LIN {X -0.054,Y -673.462,Z 1135.531,A 0.000,B 0.000,C 90.000,E1 131.595} C_DIS
LIN {X -0.295,Y -677.512,Z 1135.522,A 0.000,B 0.000,C 90.000,E1 129.930} C_DIS
LIN {X -0.323,Y -682.386,Z 1135.511,A 0.000,B 0.000,C 90.000,E1 128.016} C_DIS
LIN {X 0.074,Y -685.376,Z 1135.505,A 0.000,B 0.000,C 90.000,E1 126.790} C_DIS
LIN {X -0.070,Y -687.830,Z 1135.499,A 0.000,B 0.000,C 90.000,E1 125.851} C_DIS
LIN {X 0.211,Y -691.281,Z 1135.491,A 0.000,B 0.000,C 90.000,E1 124.405} C_DIS
LIN {X -0.010,Y -694.725,Z 1135.483,A 0.000,B 0.000,C 90.000,E1 123.007} C_DIS
LIN {X 0.378,Y -697.379,Z 1135.477,A 0.000,B 0.000,C 90.000,E1 121.799} C_DIS
LIN {X 0.197,Y -699.151,Z 1135.472,A 0.000,B 0.000,C 90.000,E1 120.875} C_DIS
LIN {X -0.296,Y -701.217,Z 1135.465,A 0.000,B 0.000,C 90.000,E1 119.745} C_DIS
LIN {X 0.133,Y -703.611,Z 1135.457,A 0.000,B 0.000,C 90.000,E1 118.309} C_DIS
LIN {X -0.259,Y -704.683,Z 1135.453,A 0.000,B 0.000,C 90.000,E1 117.641} C_DIS
LIN {X -0.025,Y -705.467,Z 1135.450,A 0.000,B 0.000,C 90.000,E1 116.924} C_DIS
LIN {X -0.153,Y -706.164,Z 1135.443,A 0.000,B 0.000,C 90.000,E1 115.771} C_DIS
LIN {X -0.220,Y -706.290,Z 1135.439,A 0.000,B 0.000,C 90.000,E1 115.079} C_DIS
LIN {X 0.068,Y -706.168,Z 1135.437,A 0.000,B 0.000,C 90.000,E1 114.591} C_DIS
LIN {X 0.006,Y -705.430,Z 1135.434,A 0.000,B 0.000,C 90.000,E1 114.131} C_DIS
LIN {X 0.008,Y -704.956,Z 1135.433,A 0.000,B 0.000,C 90.000,E1 113.898} C_DIS
LIN {X -0.206,Y -702.429,Z 1135.430,A 0.000,B 0.000,C 90.000,E1 113.334} C_DIS
LIN {X -0.066,Y -701.628,Z 1135.429,A 0.000,B 0.000,C 90.000,E1 113.206} C_DIS
LIN {X 0.201,Y -697.281,Z 1135.426,A 0.000,B 0.000,C 90.000,E1 112.717} C_DIS
LIN {X -0.312,Y -695.828,Z 1135.426,A 0.000,B 0.000,C 90.000,E1 112.642} C_DIS
LIN {X -0.182,Y -693.351,Z 1135.425,A 0.000,B 0.000,C 90.000,E1 112.514} C_DIS
LIN {X 0.282,Y -685.424,Z 1135.424,A 0.000,B 0.000,C 90.000,E1 112.206} C_DIS
LIN {X -0.173,Y -682.533,Z 1135.423,A 0.000,B 0.000,C 90.000,E1 112.206} C_DIS
LIN {X -0.220,Y -676.235,Z 1135.423,A 0.000,B 0.000,C 90.000,E1 112.153} C_DIS
LIN {X -0.243,Y -603.153,Z 1135.423,A 0.000,B 0.000,C 90.000,E1 112.153} C_DIS
LIN {X 0.311,Y -600.036,Z 1135.422,A 0.000,B 0.000,C 90.000,E1 111.897} C_DIS
LIN {X -0.184,Y -595.483,Z 1135.420,A 0.000,B 0.000,C 90.000,E1 111.589} C_DIS
LIN {X -0.037,Y -584.010,Z 1135.414,A 0.000,B 0.000,C 90.000,E1 110.556} C_DIS
LIN {X 0.171,Y -575.780,Z 1135.410,A 0.000,B 0.000,C 90.000,E1 109.812} C_DIS
LIN {X -0.325,Y -569.798,Z 1135.408,A 0.000,B 0.000,C 90.000,E1 109.396} C_DIS
LIN {X -0.170,Y -568.295,Z 1135.407,A 0.000,B 0.000,C 90.000,E1 109.268} C_DIS
LIN {X 0.057,Y -560.118,Z 1135.404,A 0.000,B 0.000,C 90.000,E1 108.725} C_DIS
LIN {X 0.230,Y -555.289,Z 1135.402,A 0.000,B 0.000,C 90.000,E1 108.417} C_DIS
LIN {X -0.209,Y -550.970,Z 1135.401,A 0.000,B 0.000,C 90.000,E1 108.127} C_DIS
LIN {X 0.260,Y -549.678,Z 1135.400,A 0.000,B 0.000,C 90.000,E1 107.873} C_DIS
LIN {X 0.219,Y -549.656,Z 1135.399,A 0.000,B 0.000,C 90.000,E1 107.873} C_DIS
LIN {X 0.011,Y -549.420,Z 1135.397,A 0.000,B 0.000,C 90.000,E1 107.457} C_DIS
LIN {X 0.002,Y -551.243,Z 1135.381,A 0.000,B 0.000,C 90.000,E1 104.662} C_DIS
LIN {X -0.248,Y -552.639,Z 1135.372,A 0.000,B 0.000,C 90.000,E1 103.008} C_DIS
LIN {X 0.058,Y -554.057,Z 1135.363,A 0.000,B 0.000,C 90.000,E1 101.299} C_DIS
LIN {X 0.043,Y -555.316,Z 1135.355,A 0.000,B 0.000,C 90.000,E1 99.905} C_DIS
LIN {X 0.186,Y -556.857,Z 1135.346,A 0.000,B 0.000,C 90.000,E1 98.219} C_DIS
LIN {X 0.142,Y -558.055,Z 1135.338,A 0.000,B 0.000,C 90.000,E1 96.834} C_DIS
LIN {X 0.193,Y -559.539,Z 1135.329,A 0.000,B 0.000,C 90.000,E1 95.163} C_DIS
LIN {X 0.140,Y -560.678,Z 1135.321,A 0.000,B 0.000,C 90.000,E1 93.784} C_DIS
LIN {X 0.072,Y -561.691,Z 1135.313,A 0.000,B 0.000,C 90.000,E1 92.407} C_DIS
LIN {X 0.022,Y -562.668,Z 1135.306,A 0.000,B 0.000,C 90.000,E1 91.031} C_DIS
LIN {X 0.081,Y -563.758,Z 1135.297,A 0.000,B 0.000,C 90.000,E1 89.370} C_DIS
LIN {X -0.164,Y -564.194,Z 1135.292,A 0.000,B 0.000,C 90.000,E1 88.568} C_DIS
LIN {X -0.067,Y -565.185,Z 1135.283,A 0.000,B 0.000,C 90.000,E1 86.906} C_DIS
LIN {X -0.026,Y -565.914,Z 1135.275,A 0.000,B 0.000,C 90.000,E1 85.527} C_DIS
LIN {X 0.031,Y -566.496,Z 1135.268,A 0.000,B 0.000,C 90.000,E1 84.147} C_DIS
LIN {X -0.236,Y -567.248,Z 1135.258,A 0.000,B 0.000,C 90.000,E1 82.527} C_DIS
LIN {X -0.092,Y -567.901,Z 1135.251,A 0.000,B 0.000,C 90.000,E1 81.141} C_DIS
LIN {X -0.235,Y -568.620,Z 1135.242,A 0.000,B 0.000,C 90.000,E1 79.511} C_DIS
LIN {X -0.186,Y -569.504,Z 1135.231,A 0.000,B 0.000,C 90.000,E1 77.589} C_DIS
LIN {X -0.063,Y -570.280,Z 1135.222,A 0.000,B 0.000,C 90.000,E1 75.936} C_DIS
LIN {X 0.045,Y -571.479,Z 1135.210,A 0.000,B 0.000,C 90.000,E1 73.740} C_DIS
LIN {X 0.181,Y -572.362,Z 1135.202,A 0.000,B 0.000,C 90.000,E1 72.362} C_DIS
LIN {X 0.142,Y -573.611,Z 1135.193,A 0.000,B 0.000,C 90.000,E1 70.732} C_DIS
LIN {X 0.152,Y -575.711,Z 1135.179,A 0.000,B 0.000,C 90.000,E1 68.284} C_DIS
LIN {X 0.208,Y -577.022,Z 1135.172,A 0.000,B 0.000,C 90.000,E1 66.922} C_DIS
LIN {X 0.130,Y -578.428,Z 1135.163,A 0.000,B 0.000,C 90.000,E1 65.305} C_DIS
LIN {X -0.306,Y -579.211,Z 1135.158,A 0.000,B 0.000,C 90.000,E1 64.537} C_DIS
LIN {X 0.151,Y -580.566,Z 1135.149,A 0.000,B 0.000,C 90.000,E1 62.871} C_DIS
LIN {X 0.119,Y -581.934,Z 1135.140,A 0.000,B 0.000,C 90.000,E1 61.257} C_DIS
LIN {X -0.114,Y -583.067,Z 1135.131,A 0.000,B 0.000,C 90.000,E1 59.665} C_DIS
LIN {X -0.189,Y -583.979,Z 1135.124,A 0.000,B 0.000,C 90.000,E1 58.329} C_DIS
LIN {X -0.078,Y -584.923,Z 1135.115,A 0.000,B 0.000,C 90.000,E1 56.707} C_DIS
LIN {X -0.113,Y -585.846,Z 1135.106,A 0.000,B 0.000,C 90.000,E1 55.102} C_DIS
LIN {X -0.131,Y -586.745,Z 1135.097,A 0.000,B 0.000,C 90.000,E1 53.497} C_DIS
LIN {X -0.019,Y -587.109,Z 1135.093,A 0.000,B 0.000,C 90.000,E1 52.683} C_DIS
LIN {X 0.064,Y -587.974,Z 1135.082,A 0.000,B 0.000,C 90.000,E1 50.803} C_DIS
LIN {X -0.061,Y -588.254,Z 1135.076,A 0.000,B 0.000,C 90.000,E1 49.747} C_DIS
LIN {X -0.179,Y -588.386,Z 1135.070,A 0.000,B 0.000,C 90.000,E1 48.690} C_DIS
LIN {X 0.216,Y -588.248,Z 1135.060,A 0.000,B 0.000,C 90.000,E1 46.782} C_DIS
LIN {X -0.188,Y -587.888,Z 1135.053,A 0.000,B 0.000,C 90.000,E1 45.486} C_DIS
LIN {X -0.345,Y -587.498,Z 1135.047,A 0.000,B 0.000,C 90.000,E1 44.433} C_DIS
LIN {X -0.086,Y -586.841,Z 1135.041,A 0.000,B 0.000,C 90.000,E1 43.338} C_DIS
LIN {X 0.242,Y -586.545,Z 1135.038,A 0.000,B 0.000,C 90.000,E1 42.771} C_DIS
LIN {X 0.169,Y -585.976,Z 1135.035,A 0.000,B 0.000,C 90.000,E1 42.243} C_DIS
LIN {X -0.086,Y -585.834,Z 1135.033,A 0.000,B 0.000,C 90.000,E1 42.000} C_DIS
LIN {X 0.058,Y -583.950,Z 1135.024,A 0.000,B 0.000,C 90.000,E1 40.378} C_DIS
LIN {X -0.033,Y -583.350,Z 1135.021,A 0.000,B 0.000,C 90.000,E1 39.850} C_DIS
LIN {X -0.059,Y -581.407,Z 1135.014,A 0.000,B 0.000,C 90.000,E1 38.508} C_DIS
LIN {X -0.023,Y -579.036,Z 1135.006,A 0.000,B 0.000,C 90.000,E1 37.156} C_DIS
LIN {X -0.339,Y -577.328,Z 1135.002,A 0.000,B 0.000,C 90.000,E1 36.377} C_DIS
LIN {X 0.134,Y -575.314,Z 1134.997,A 0.000,B 0.000,C 90.000,E1 35.518} C_DIS
LIN {X 0.103,Y -573.841,Z 1134.994,A 0.000,B 0.000,C 90.000,E1 34.978} C_DIS
LIN {X -0.265,Y -571.310,Z 1134.990,A 0.000,B 0.000,C 90.000,E1 34.199} C_DIS
LIN {X 0.001,Y -569.465,Z 1134.987,A 0.000,B 0.000,C 90.000,E1 33.627} C_DIS
LIN {X -0.142,Y -565.241,Z 1134.981,A 0.000,B 0.000,C 90.000,E1 32.546} C_DIS
LIN {X -0.331,Y -562.292,Z 1134.977,A 0.000,B 0.000,C 90.000,E1 31.878} C_DIS
LIN {X 0.190,Y -556.954,Z 1134.971,A 0.000,B 0.000,C 90.000,E1 30.718} C_DIS
LIN {X 0.176,Y -551.709,Z 1134.965,A 0.000,B 0.000,C 90.000,E1 29.745} C_DIS
LIN {X -0.254,Y -546.846,Z 1134.961,A 0.000,B 0.000,C 90.000,E1 28.949} C_DIS
LIN {X 0.094,Y -540.592,Z 1134.955,A 0.000,B 0.000,C 90.000,E1 27.924} C_DIS
LIN {X 0.024,Y -534.510,Z 1134.950,A 0.000,B 0.000,C 90.000,E1 27.078} C_DIS
LIN {X 0.033,Y -529.067,Z 1134.947,A 0.000,B 0.000,C 90.000,E1 26.360} C_DIS
LIN {X -0.208,Y -523.297,Z 1134.943,A 0.000,B 0.000,C 90.000,E1 25.668} C_DIS
LIN {X -0.110,Y -514.407,Z 1134.937,A 0.000,B 0.000,C 90.000,E1 24.643} C_DIS
LIN {X 0.110,Y -507.754,Z 1134.933,A 0.000,B 0.000,C 90.000,E1 23.898} C_DIS
LIN {X -0.063,Y -499.557,Z 1134.928,A 0.000,B 0.000,C 90.000,E1 23.078} C_DIS
LIN {X -0.207,Y -491.090,Z 1134.924,A 0.000,B 0.000,C 90.000,E1 22.280} C_DIS
LIN {X 0.040,Y -483.962,Z 1134.920,A 0.000,B 0.000,C 90.000,E1 21.589} C_DIS
LIN {X 0.239,Y -475.392,Z 1134.916,A 0.000,B 0.000,C 90.000,E1 20.791} C_DIS
LIN {X -0.073,Y -468.011,Z 1134.912,A 0.000,B 0.000,C 90.000,E1 20.174} C_DIS
LIN {X 0.109,Y -453.457,Z 1134.905,A 0.000,B 0.000,C 90.000,E1 18.852} C_DIS
LIN {X 0.049,Y -437.348,Z 1134.896,A 0.000,B 0.000,C 90.000,E1 17.347} C_DIS
LIN {X -0.102,Y -423.156,Z 1134.888,A 0.000,B 0.000,C 90.000,E1 15.898} C_DIS
LIN {X 0.159,Y -412.057,Z 1134.881,A 0.000,B 0.000,C 90.000,E1 14.592} C_DIS
LIN {X 0.188,Y -404.239,Z 1134.876,A 0.000,B 0.000,C 90.000,E1 13.592} C_DIS
LIN {X 0.056,Y -399.562,Z 1134.872,A 0.000,B 0.000,C 90.000,E1 12.939} C_DIS
LIN {X 0.041,Y -397.373,Z 1134.870,A 0.000,B 0.000,C 90.000,E1 12.591} C_DIS
LIN {X -0.181,Y -394.183,Z 1134.867,A 0.000,B 0.000,C 90.000,E1 12.007} C_DIS
LIN {X 0.121,Y -392.964,Z 1134.865,A 0.000,B 0.000,C 90.000,E1 11.591} C_DIS
LIN {X 0.063,Y -392.555,Z 1134.864,A 0.000,B 0.000,C 90.000,E1 11.422} C_DIS
LIN {X 0.051,Y -392.145,Z 1134.862,A 0.000,B 0.000,C 90.000,E1 11.074} C_DIS
LIN {X 0.065,Y -392.473,Z 1134.859,A 0.000,B 0.000,C 90.000,E1 10.546} C_DIS
LIN {X 0.077,Y -392.640,Z 1134.858,A 0.000,B 0.000,C 90.000,E1 10.366} C_DIS
LIN {X -0.078,Y -394.573,Z 1134.852,A 0.000,B 0.000,C 90.000,E1 9.434} C_DIS
LIN {X 0.146,Y -397.451,Z 1134.847,A 0.000,B 0.000,C 90.000,E1 8.341} C_DIS
LIN {X -0.003,Y -402.854,Z 1134.837,A 0.000,B 0.000,C 90.000,E1 6.606} C_DIS
LIN {X -0.036,Y -404.749,Z 1134.834,A 0.000,B 0.000,C 90.000,E1 6.087} C_DIS
LIN {X -0.057,Y -407.334,Z 1134.831,A 0.000,B 0.000,C 90.000,E1 5.568} C_DIS
LIN {X -0.034,Y -408.383,Z 1134.830,A 0.000,B 0.000,C 90.000,E1 5.391} C_DIS
LIN {X -0.051,Y -411.120,Z 1134.828,A 0.000,B 0.000,C 90.000,E1 5.049} C_DIS
LIN {X -0.052,Y -412.815,Z 1134.827,A 0.000,B 0.000,C 90.000,E1 4.878} C_DIS
LIN {X -0.122,Y -416.366,Z 1134.825,A 0.000,B 0.000,C 90.000,E1 4.588} C_DIS
LIN {X 0.180,Y -423.924,Z 1134.823,A 0.000,B 0.000,C 90.000,E1 4.012} C_DIS
LIN {X 0.208,Y -446.765,Z 1134.814,A 0.000,B 0.000,C 90.000,E1 2.407} C_DIS
LIN {X 0.220,Y -463.099,Z 1134.807,A 0.000,B 0.000,C 90.000,E1 1.318} C_DIS
LIN {X -0.195,Y -474.343,Z 1134.803,A 0.000,B 0.000,C 90.000,E1 0.630} C_DIS
LIN {X 0.000,Y -483.330,Z 1134.800,A 0.000,B 0.000,C 90.000,E1 360.000} C_DIS
LIN {X 0.238,Y -490.911,Z 1134.797,A 0.000,B 0.000,C 90.000,E1 359.427} C_DIS
LIN {X -0.246,Y -496.999,Z 1134.794,A 0.000,B 0.000,C 90.000,E1 359.026} C_DIS
LIN {X 0.117,Y -502.993,Z 1134.792,A 0.000,B 0.000,C 90.000,E1 358.511} C_DIS
LIN {X 0.177,Y -510.196,Z 1134.788,A 0.000,B 0.000,C 90.000,E1 357.879} C_DIS
LIN {X 0.038,Y -517.140,Z 1134.785,A 0.000,B 0.000,C 90.000,E1 357.249} C_DIS
LIN {X 0.060,Y -521.102,Z 1134.783,A 0.000,B 0.000,C 90.000,E1 356.846} C_DIS
LIN {X -0.041,Y -527.440,Z 1134.779,A 0.000,B 0.000,C 90.000,E1 356.159} C_DIS
LIN {X 0.024,Y -532.263,Z 1134.776,A 0.000,B 0.000,C 90.000,E1 355.584} C_DIS
LIN {X -0.240,Y -537.755,Z 1134.771,A 0.000,B 0.000,C 90.000,E1 354.894} C_DIS
LIN {X 0.081,Y -542.573,Z 1134.768,A 0.000,B 0.000,C 90.000,E1 354.147} C_DIS
LIN {X -0.035,Y -546.969,Z 1134.764,A 0.000,B 0.000,C 90.000,E1 353.451} C_DIS
LIN {X 0.084,Y -550.174,Z 1134.760,A 0.000,B 0.000,C 90.000,E1 352.875} C_DIS
LIN {X 0.088,Y -555.222,Z 1134.755,A 0.000,B 0.000,C 90.000,E1 351.894} C_DIS
LIN {X -0.292,Y -557.758,Z 1134.752,A 0.000,B 0.000,C 90.000,E1 351.376} C_DIS
LIN {X -0.269,Y -560.636,Z 1134.748,A 0.000,B 0.000,C 90.000,E1 350.679} C_DIS
LIN {X 0.181,Y -563.777,Z 1134.744,A 0.000,B 0.000,C 90.000,E1 349.803} C_DIS
LIN {X 0.011,Y -566.665,Z 1134.739,A 0.000,B 0.000,C 90.000,E1 348.993} C_DIS
LIN {X 0.156,Y -570.210,Z 1134.733,A 0.000,B 0.000,C 90.000,E1 347.881} C_DIS
LIN {X 0.119,Y -574.235,Z 1134.725,A 0.000,B 0.000,C 90.000,E1 346.520} C_DIS
LIN {X 0.018,Y -577.923,Z 1134.718,A 0.000,B 0.000,C 90.000,E1 345.172} C_DIS
LIN {X 0.275,Y -581.457,Z 1134.710,A 0.000,B 0.000,C 90.000,E1 343.795} C_DIS
LIN {X 0.271,Y -585.478,Z 1134.701,A 0.000,B 0.000,C 90.000,E1 342.181} C_DIS
LIN {X 0.016,Y -587.351,Z 1134.697,A 0.000,B 0.000,C 90.000,E1 341.402} C_DIS
LIN {X 0.197,Y -589.644,Z 1134.691,A 0.000,B 0.000,C 90.000,E1 340.315} C_DIS
LIN {X 0.058,Y -591.720,Z 1134.685,A 0.000,B 0.000,C 90.000,E1 339.263} C_DIS
LIN {X -0.263,Y -593.666,Z 1134.679,A 0.000,B 0.000,C 90.000,E1 338.230} C_DIS
LIN {X -0.016,Y -594.827,Z 1134.675,A 0.000,B 0.000,C 90.000,E1 337.411} C_DIS
LIN {X -0.167,Y -596.352,Z 1134.667,A 0.000,B 0.000,C 90.000,E1 336.102} C_DIS
LIN {X -0.216,Y -597.148,Z 1134.661,A 0.000,B 0.000,C 90.000,E1 335.049} C_DIS
LIN {X 0.072,Y -597.559,Z 1134.657,A 0.000,B 0.000,C 90.000,E1 334.229} C_DIS
LIN {X 0.093,Y -597.595,Z 1134.652,A 0.000,B 0.000,C 90.000,E1 333.435} C_DIS
LIN {X -0.145,Y -597.263,Z 1134.648,A 0.000,B 0.000,C 90.000,E1 332.666} C_DIS
LIN {X 0.137,Y -596.685,Z 1134.644,A 0.000,B 0.000,C 90.000,E1 331.847} C_DIS
LIN {X 0.252,Y -596.143,Z 1134.641,A 0.000,B 0.000,C 90.000,E1 331.307} C_DIS
LIN {X -0.012,Y -595.032,Z 1134.636,A 0.000,B 0.000,C 90.000,E1 330.539} C_DIS
LIN {X 0.203,Y -592.887,Z 1134.630,A 0.000,B 0.000,C 90.000,E1 329.459} C_DIS
LIN {X -0.001,Y -591.481,Z 1134.628,A 0.000,B 0.000,C 90.000,E1 328.948} C_DIS
LIN {X 0.087,Y -589.792,Z 1134.625,A 0.000,B 0.000,C 90.000,E1 328.408} C_DIS
LIN {X 0.164,Y -587.964,Z 1134.622,A 0.000,B 0.000,C 90.000,E1 327.867} C_DIS
LIN {X -0.076,Y -584.644,Z 1134.617,A 0.000,B 0.000,C 90.000,E1 327.089} C_DIS
LIN {X -0.107,Y -581.397,Z 1134.613,A 0.000,B 0.000,C 90.000,E1 326.421} C_DIS
LIN {X 0.070,Y -576.825,Z 1134.609,A 0.000,B 0.000,C 90.000,E1 325.595} C_DIS
LIN {X 0.048,Y -573.585,Z 1134.606,A 0.000,B 0.000,C 90.000,E1 325.055} C_DIS
LIN {X -0.232,Y -569.139,Z 1134.602,A 0.000,B 0.000,C 90.000,E1 324.402} C_DIS
LIN {X -0.205,Y -566.307,Z 1134.600,A 0.000,B 0.000,C 90.000,E1 323.989} C_DIS
LIN {X 0.027,Y -562.124,Z 1134.597,A 0.000,B 0.000,C 90.000,E1 323.417} C_DIS
LIN {X -0.254,Y -554.221,Z 1134.591,A 0.000,B 0.000,C 90.000,E1 322.477} C_DIS
LIN {X -0.053,Y -546.776,Z 1134.587,A 0.000,B 0.000,C 90.000,E1 321.618} C_DIS
LIN {X -0.142,Y -536.796,Z 1134.581,A 0.000,B 0.000,C 90.000,E1 320.517} C_DIS
LIN {X -0.018,Y -533.738,Z 1134.578,A 0.000,B 0.000,C 90.000,E1 320.114} C_DIS
LIN {X 0.064,Y -530.380,Z 1134.576,A 0.000,B 0.000,C 90.000,E1 319.585} C_DIS
LIN {X -0.124,Y -527.923,Z 1134.573,A 0.000,B 0.000,C 90.000,E1 319.094} C_DIS
LIN {X -0.183,Y -526.213,Z 1134.570,A 0.000,B 0.000,C 90.000,E1 318.609} C_DIS
LIN {X 0.088,Y -525.373,Z 1134.568,A 0.000,B 0.000,C 90.000,E1 318.243} C_DIS
LIN {X -0.190,Y -524.466,Z 1134.566,A 0.000,B 0.000,C 90.000,E1 317.838} C_DIS
LIN {X 0.222,Y -523.768,Z 1134.562,A 0.000,B 0.000,C 90.000,E1 317.067} C_DIS
LIN {X 0.338,Y -523.606,Z 1134.555,A 0.000,B 0.000,C 90.000,E1 315.891} C_DIS
LIN {X -0.056,Y -523.818,Z 1134.546,A 0.000,B 0.000,C 90.000,E1 314.190} C_DIS
LIN {X 0.182,Y -524.344,Z 1134.533,A 0.000,B 0.000,C 90.000,E1 311.838} C_DIS
LIN {X -0.264,Y -525.395,Z 1134.520,A 0.000,B 0.000,C 90.000,E1 309.564} C_DIS
LIN {X -0.198,Y -526.773,Z 1134.507,A 0.000,B 0.000,C 90.000,E1 307.237} C_DIS
LIN {X 0.068,Y -527.900,Z 1134.497,A 0.000,B 0.000,C 90.000,E1 305.471} C_DIS
LIN {X 0.038,Y -529.291,Z 1134.486,A 0.000,B 0.000,C 90.000,E1 303.452} C_DIS
LIN {X 0.165,Y -530.963,Z 1134.473,A 0.000,B 0.000,C 90.000,E1 301.131} C_DIS
LIN {X -0.033,Y -531.827,Z 1134.467,A 0.000,B 0.000,C 90.000,E1 300.001} C_DIS
LIN {X -0.046,Y -532.818,Z 1134.459,A 0.000,B 0.000,C 90.000,E1 298.565} C_DIS
LIN {X 0.243,Y -533.431,Z 1134.452,A 0.000,B 0.000,C 90.000,E1 297.385} C_DIS
LIN {X 0.294,Y -533.863,Z 1134.446,A 0.000,B 0.000,C 90.000,E1 296.232} C_DIS
LIN {X 0.121,Y -534.113,Z 1134.440,A 0.000,B 0.000,C 90.000,E1 295.103} C_DIS
LIN {X -0.111,Y -534.178,Z 1134.432,A 0.000,B 0.000,C 90.000,E1 293.695} C_DIS
LIN {X -0.083,Y -534.166,Z 1134.424,A 0.000,B 0.000,C 90.000,E1 292.259} C_DIS
LIN {X -0.168,Y -534.153,Z 1134.419,A 0.000,B 0.000,C 90.000,E1 291.408} C_DIS
LIN {X 0.162,Y -534.029,Z 1134.411,A 0.000,B 0.000,C 90.000,E1 289.939} C_DIS
LIN {X 0.003,Y -533.695,Z 1134.401,A 0.000,B 0.000,C 90.000,E1 288.236} C_DIS
LIN {X 0.171,Y -533.179,Z 1134.392,A 0.000,B 0.000,C 90.000,E1 286.496} C_DIS
LIN {X 0.139,Y -532.563,Z 1134.384,A 0.000,B 0.000,C 90.000,E1 285.064} C_DIS
LIN {X 0.037,Y -531.559,Z 1134.373,A 0.000,B 0.000,C 90.000,E1 283.063} C_DIS
LIN {X -0.236,Y -530.643,Z 1134.363,A 0.000,B 0.000,C 90.000,E1 281.366} C_DIS
LIN {X -0.046,Y -529.777,Z 1134.355,A 0.000,B 0.000,C 90.000,E1 279.905} C_DIS
LIN {X 0.035,Y -529.001,Z 1134.347,A 0.000,B 0.000,C 90.000,E1 278.454} C_DIS
LIN {X 0.070,Y -527.954,Z 1134.336,A 0.000,B 0.000,C 90.000,E1 276.429} C_DIS
LIN {X -0.040,Y -527.048,Z 1134.325,A 0.000,B 0.000,C 90.000,E1 274.416} C_DIS
LIN {X -0.173,Y -526.285,Z 1134.315,A 0.000,B 0.000,C 90.000,E1 272.694} C_DIS
LIN {X 0.208,Y -525.681,Z 1134.307,A 0.000,B 0.000,C 90.000,E1 271.203} C_DIS
LIN {X 0.043,Y -525.038,Z 1134.299,A 0.000,B 0.000,C 90.000,E1 269.771} C_DIS
LIN {X -0.137,Y -524.363,Z 1134.291,A 0.000,B 0.000,C 90.000,E1 268.339} C_DIS
LIN {X 0.204,Y -523.639,Z 1134.283,A 0.000,B 0.000,C 90.000,E1 266.849} C_DIS
LIN {X 0.031,Y -522.676,Z 1134.273,A 0.000,B 0.000,C 90.000,E1 265.122} C_DIS
LIN {X -0.081,Y -522.115,Z 1134.268,A 0.000,B 0.000,C 90.000,E1 264.261} C_DIS
LIN {X -0.148,Y -521.326,Z 1134.263,A 0.000,B 0.000,C 90.000,E1 263.394} C_DIS
LIN {X 0.217,Y -519.659,Z 1134.254,A 0.000,B 0.000,C 90.000,E1 261.602} C_DIS
LIN {X 0.002,Y -517.601,Z 1134.242,A 0.000,B 0.000,C 90.000,E1 259.577} C_DIS
LIN {X -0.058,Y -516.139,Z 1134.234,A 0.000,B 0.000,C 90.000,E1 258.117} C_DIS
LIN {X -0.055,Y -514.399,Z 1134.224,A 0.000,B 0.000,C 90.000,E1 256.353} C_DIS
LIN {X 0.038,Y -512.873,Z 1134.214,A 0.000,B 0.000,C 90.000,E1 254.574} C_DIS
LIN {X 0.239,Y -511.161,Z 1134.204,A 0.000,B 0.000,C 90.000,E1 252.779} C_DIS
LIN {X -0.090,Y -509.365,Z 1134.195,A 0.000,B 0.000,C 90.000,E1 251.040} C_DIS
LIN {X -0.227,Y -507.727,Z 1134.186,A 0.000,B 0.000,C 90.000,E1 249.571} C_DIS
LIN {X 0.078,Y -506.094,Z 1134.178,A 0.000,B 0.000,C 90.000,E1 248.050} C_DIS
LIN {X 0.061,Y -504.340,Z 1134.170,A 0.000,B 0.000,C 90.000,E1 246.561} C_DIS
LIN {X -0.242,Y -502.431,Z 1134.162,A 0.000,B 0.000,C 90.000,E1 245.101} C_DIS
LIN {X -0.122,Y -500.332,Z 1134.153,A 0.000,B 0.000,C 90.000,E1 243.589} C_DIS
LIN {X -0.273,Y -498.126,Z 1134.145,A 0.000,B 0.000,C 90.000,E1 242.103} C_DIS
LIN {X -0.223,Y -495.774,Z 1134.136,A 0.000,B 0.000,C 90.000,E1 240.589} C_DIS
LIN {X -0.217,Y -493.289,Z 1134.128,A 0.000,B 0.000,C 90.000,E1 239.076} C_DIS
LIN {X -0.172,Y -490.326,Z 1134.118,A 0.000,B 0.000,C 90.000,E1 237.248} C_DIS
LIN {X 0.073,Y -487.286,Z 1134.108,A 0.000,B 0.000,C 90.000,E1 235.388} C_DIS
LIN {X 0.015,Y -484.744,Z 1134.099,A 0.000,B 0.000,C 90.000,E1 233.863} C_DIS
LIN {X -0.198,Y -482.045,Z 1134.091,A 0.000,B 0.000,C 90.000,E1 232.351} C_DIS
LIN {X -0.080,Y -480.518,Z 1134.086,A 0.000,B 0.000,C 90.000,E1 231.412} C_DIS
LIN {X 0.027,Y -477.121,Z 1134.075,A 0.000,B 0.000,C 90.000,E1 229.542} C_DIS
LIN {X 0.018,Y -473.849,Z 1134.065,A 0.000,B 0.000,C 90.000,E1 227.676} C_DIS
LIN {X 0.026,Y -469.997,Z 1134.053,A 0.000,B 0.000,C 90.000,E1 225.486} C_DIS
LIN {X -0.156,Y -467.007,Z 1134.042,A 0.000,B 0.000,C 90.000,E1 223.623} C_DIS
LIN {X 0.266,Y -464.315,Z 1134.032,A 0.000,B 0.000,C 90.000,E1 221.676} C_DIS
LIN {X -0.200,Y -461.059,Z 1134.018,A 0.000,B 0.000,C 90.000,E1 219.197} C_DIS
LIN {X 0.050,Y -457.876,Z 1134.002,A 0.000,B 0.000,C 90.000,E1 216.297} C_DIS
LIN {X 0.097,Y -456.223,Z 1133.993,A 0.000,B 0.000,C 90.000,E1 214.692} C_DIS
LIN {X -0.064,Y -453.494,Z 1133.973,A 0.000,B 0.000,C 90.000,E1 211.180} C_DIS
LIN {X 0.275,Y -452.576,Z 1133.963,A 0.000,B 0.000,C 90.000,E1 209.205} C_DIS
LIN {X -0.018,Y -452.255,Z 1133.952,A 0.000,B 0.000,C 90.000,E1 207.308} C_DIS
LIN {X 0.283,Y -452.928,Z 1133.941,A 0.000,B 0.000,C 90.000,E1 205.335} C_DIS
LIN {X -0.076,Y -454.354,Z 1133.932,A 0.000,B 0.000,C 90.000,E1 203.770} C_DIS
LIN {X 0.017,Y -456.817,Z 1133.923,A 0.000,B 0.000,C 90.000,E1 202.153} C_DIS
LIN {X -0.009,Y -459.940,Z 1133.914,A 0.000,B 0.000,C 90.000,E1 200.556} C_DIS
LIN {X -0.055,Y -464.584,Z 1133.904,A 0.000,B 0.000,C 90.000,E1 198.652} C_DIS
LIN {X -0.044,Y -471.259,Z 1133.891,A 0.000,B 0.000,C 90.000,E1 196.441} C_DIS
LIN {X 0.196,Y -477.658,Z 1133.881,A 0.000,B 0.000,C 90.000,E1 194.537} C_DIS
LIN {X 0.076,Y -487.836,Z 1133.865,A 0.000,B 0.000,C 90.000,E1 191.771} C_DIS
LIN {X -0.205,Y -496.098,Z 1133.854,A 0.000,B 0.000,C 90.000,E1 189.670} C_DIS
LIN {X -0.137,Y -500.906,Z 1133.847,A 0.000,B 0.000,C 90.000,E1 188.454} C_DIS
LIN {X -0.057,Y -506.934,Z 1133.839,A 0.000,B 0.000,C 90.000,E1 186.947} C_DIS
LIN {X 0.011,Y -512.803,Z 1133.830,A 0.000,B 0.000,C 90.000,E1 185.454} C_DIS
LIN {X 0.241,Y -518.665,Z 1133.822,A 0.000,B 0.000,C 90.000,E1 183.955} C_DIS
LIN {X 0.232,Y -525.249,Z 1133.813,A 0.000,B 0.000,C 90.000,E1 182.350} C_DIS
LIN {X -0.180,Y -531.662,Z 1133.804,A 0.000,B 0.000,C 90.000,E1 180.802} C_DIS
LIN {X 0.078,Y -540.459,Z 1133.792,A 0.000,B 0.000,C 90.000,E1 178.625} C_DIS
LIN {X -0.101,Y -544.524,Z 1133.787,A 0.000,B 0.000,C 90.000,E1 177.650} C_DIS
LIN {X 0.252,Y -552.798,Z 1133.776,A 0.000,B 0.000,C 90.000,E1 175.641} C_DIS
LIN {X 0.102,Y -558.621,Z 1133.768,A 0.000,B 0.000,C 90.000,E1 174.261} C_DIS
LIN {X 0.196,Y -565.641,Z 1133.759,A 0.000,B 0.000,C 90.000,E1 172.591} C_DIS
LIN {X -0.060,Y -572.638,Z 1133.750,A 0.000,B 0.000,C 90.000,E1 170.971} C_DIS
LIN {X 0.167,Y -577.221,Z 1133.744,A 0.000,B 0.000,C 90.000,E1 169.859} C_DIS
LIN {X 0.252,Y -583.800,Z 1133.735,A 0.000,B 0.000,C 90.000,E1 168.229} C_DIS
LIN {X -0.243,Y -589.145,Z 1133.727,A 0.000,B 0.000,C 90.000,E1 166.937} C_DIS
LIN {X -0.040,Y -592.217,Z 1133.723,A 0.000,B 0.000,C 90.000,E1 166.117} C_DIS
LIN {X 0.042,Y -596.185,Z 1133.717,A 0.000,B 0.000,C 90.000,E1 165.046} C_DIS
LIN {X 0.184,Y -599.927,Z 1133.711,A 0.000,B 0.000,C 90.000,E1 163.976} C_DIS
LIN {X 0.077,Y -602.558,Z 1133.707,A 0.000,B 0.000,C 90.000,E1 163.196} C_DIS
LIN {X 0.217,Y -606.869,Z 1133.699,A 0.000,B 0.000,C 90.000,E1 161.873} C_DIS
LIN {X -0.152,Y -610.856,Z 1133.692,A 0.000,B 0.000,C 90.000,E1 160.604} C_DIS
LIN {X -0.206,Y -613.934,Z 1133.686,A 0.000,B 0.000,C 90.000,E1 159.571} C_DIS
LIN {X -0.258,Y -617.475,Z 1133.679,A 0.000,B 0.000,C 90.000,E1 158.284} C_DIS
LIN {X -0.269,Y -621.586,Z 1133.671,A 0.000,B 0.000,C 90.000,E1 156.741} C_DIS
LIN {X 0.294,Y -624.876,Z 1133.664,A 0.000,B 0.000,C 90.000,E1 155.409} C_DIS
LIN {X 0.091,Y -628.048,Z 1133.656,A 0.000,B 0.000,C 90.000,E1 154.152} C_DIS
LIN {X 0.181,Y -630.423,Z 1133.651,A 0.000,B 0.000,C 90.000,E1 153.127} C_DIS
LIN {X -0.222,Y -633.320,Z 1133.644,A 0.000,B 0.000,C 90.000,E1 151.897} C_DIS
LIN {X 0.281,Y -636.079,Z 1133.637,A 0.000,B 0.000,C 90.000,E1 150.589} C_DIS
LIN {X 0.279,Y -638.705,Z 1133.630,A 0.000,B 0.000,C 90.000,E1 149.331} C_DIS
LIN {X -0.232,Y -641.242,Z 1133.623,A 0.000,B 0.000,C 90.000,E1 148.122} C_DIS
LIN {X -0.303,Y -644.043,Z 1133.615,A 0.000,B 0.000,C 90.000,E1 146.628} C_DIS
LIN {X 0.037,Y -646.682,Z 1133.606,A 0.000,B 0.000,C 90.000,E1 145.102} C_DIS
LIN {X -0.010,Y -648.788,Z 1133.599,A 0.000,B 0.000,C 90.000,E1 143.863} C_DIS
LIN {X 0.197,Y -651.728,Z 1133.590,A 0.000,B 0.000,C 90.000,E1 142.110} C_DIS
LIN {X 0.016,Y -655.266,Z 1133.579,A 0.000,B 0.000,C 90.000,E1 140.150} C_DIS
LIN {X -0.129,Y -657.611,Z 1133.572,A 0.000,B 0.000,C 90.000,E1 138.933} C_DIS
LIN {X -0.261,Y -660.519,Z 1133.564,A 0.000,B 0.000,C 90.000,E1 137.472} C_DIS
LIN {X 0.093,Y -664.433,Z 1133.553,A 0.000,B 0.000,C 90.000,E1 135.486} C_DIS
LIN {X 0.082,Y -669.296,Z 1133.541,A 0.000,B 0.000,C 90.000,E1 133.299} C_DIS
LIN {X 0.193,Y -673.360,Z 1133.531,A 0.000,B 0.000,C 90.000,E1 131.595} C_DIS
LIN {X -0.069,Y -676.807,Z 1133.523,A 0.000,B 0.000,C 90.000,E1 130.172} C_DIS
LIN {X -0.077,Y -682.289,Z 1133.511,A 0.000,B 0.000,C 90.000,E1 128.016} C_DIS
LIN {X -0.257,Y -684.693,Z 1133.506,A 0.000,B 0.000,C 90.000,E1 127.076} C_DIS
LIN {X -0.227,Y -687.728,Z 1133.499,A 0.000,B 0.000,C 90.000,E1 125.884} C_DIS
LIN {X -0.114,Y -691.192,Z 1133.491,A 0.000,B 0.000,C 90.000,E1 124.452} C_DIS
LIN {X -0.144,Y -694.638,Z 1133.484,A 0.000,B 0.000,C 90.000,E1 123.038} C_DIS
LIN {X 0.008,Y -696.800,Z 1133.478,A 0.000,B 0.000,C 90.000,E1 122.084} C_DIS
LIN {X 0.184,Y -698.693,Z 1133.473,A 0.000,B 0.000,C 90.000,E1 121.131} C_DIS
LIN {X -0.052,Y -701.160,Z 1133.465,A 0.000,B 0.000,C 90.000,E1 119.745} C_DIS
LIN {X -0.243,Y -703.577,Z 1133.458,A 0.000,B 0.000,C 90.000,E1 118.359} C_DIS
LIN {X -0.016,Y -704.629,Z 1133.454,A 0.000,B 0.000,C 90.000,E1 117.641} C_DIS
LIN {X -0.102,Y -705.391,Z 1133.450,A 0.000,B 0.000,C 90.000,E1 116.950} C_DIS
LIN {X -0.218,Y -706.124,Z 1133.443,A 0.000,B 0.000,C 90.000,E1 115.796} C_DIS
LIN {X 0.022,Y -706.296,Z 1133.439,A 0.000,B 0.000,C 90.000,E1 115.079} C_DIS
LIN {X -0.332,Y -706.173,Z 1133.437,A 0.000,B 0.000,C 90.000,E1 114.643} C_DIS
LIN {X -0.041,Y -705.436,Z 1133.434,A 0.000,B 0.000,C 90.000,E1 114.155} C_DIS
LIN {X 0.249,Y -704.988,Z 1133.433,A 0.000,B 0.000,C 90.000,E1 113.898} C_DIS
LIN {X 0.036,Y -702.533,Z 1133.430,A 0.000,B 0.000,C 90.000,E1 113.334} C_DIS
LIN {X 0.175,Y -701.786,Z 1133.429,A 0.000,B 0.000,C 90.000,E1 113.206} C_DIS
LIN {X -0.201,Y -697.473,Z 1133.427,A 0.000,B 0.000,C 90.000,E1 112.770} C_DIS
LIN {X -0.071,Y -696.120,Z 1133.426,A 0.000,B 0.000,C 90.000,E1 112.642} C_DIS
LIN {X 0.057,Y -693.907,Z 1133.425,A 0.000,B 0.000,C 90.000,E1 112.514} C_DIS
LIN {X 0.405,Y -685.903,Z 1133.424,A 0.000,B 0.000,C 90.000,E1 112.206} C_DIS
LIN {X -0.075,Y -683.585,Z 1133.423,A 0.000,B 0.000,C 90.000,E1 112.206} C_DIS
LIN {X -0.222,Y -676.690,Z 1133.423,A 0.000,B 0.000,C 90.000,E1 112.153} C_DIS
LIN {X -0.232,Y -603.215,Z 1133.423,A 0.000,B 0.000,C 90.000,E1 112.153} C_DIS
LIN {X 0.311,Y -600.036,Z 1133.422,A 0.000,B 0.000,C 90.000,E1 111.897} C_DIS
LIN {X -0.125,Y -595.548,Z 1133.420,A 0.000,B 0.000,C 90.000,E1 111.589} C_DIS
LIN {X 0.078,Y -582.697,Z 1133.414,A 0.000,B 0.000,C 90.000,E1 110.429} C_DIS
LIN {X -0.164,Y -574.756,Z 1133.410,A 0.000,B 0.000,C 90.000,E1 109.758} C_DIS
LIN {X 0.105,Y -568.704,Z 1133.407,A 0.000,B 0.000,C 90.000,E1 109.268} C_DIS
LIN {X -0.246,Y -560.484,Z 1133.404,A 0.000,B 0.000,C 90.000,E1 108.779} C_DIS
LIN {X 0.253,Y -554.450,Z 1133.402,A 0.000,B 0.000,C 90.000,E1 108.362} C_DIS
LIN {X -0.108,Y -550.809,Z 1133.401,A 0.000,B 0.000,C 90.000,E1 108.109} C_DIS
LIN {X 0.203,Y -549.571,Z 1133.399,A 0.000,B 0.000,C 90.000,E1 107.873} C_DIS
LIN {X 0.161,Y -549.561,Z 1133.399,A 0.000,B 0.000,C 90.000,E1 107.873} C_DIS
LIN {X -0.024,Y -549.314,Z 1133.397,A 0.000,B 0.000,C 90.000,E1 107.511} C_DIS
LIN {X -0.152,Y -550.913,Z 1133.383,A 0.000,B 0.000,C 90.000,E1 105.009} C_DIS
LIN {X 0.238,Y -552.506,Z 1133.372,A 0.000,B 0.000,C 90.000,E1 103.008} C_DIS
LIN {X -0.110,Y -553.959,Z 1133.363,A 0.000,B 0.000,C 90.000,E1 101.366} C_DIS
LIN {X 0.106,Y -555.427,Z 1133.354,A 0.000,B 0.000,C 90.000,E1 99.670} C_DIS
LIN {X 0.169,Y -556.991,Z 1133.345,A 0.000,B 0.000,C 90.000,E1 97.992} C_DIS
LIN {X 0.266,Y -558.452,Z 1133.335,A 0.000,B 0.000,C 90.000,E1 96.315} C_DIS
LIN {X 0.196,Y -559.695,Z 1133.328,A 0.000,B 0.000,C 90.000,E1 94.935} C_DIS
LIN {X 0.149,Y -560.818,Z 1133.320,A 0.000,B 0.000,C 90.000,E1 93.555} C_DIS
LIN {X 0.086,Y -561.816,Z 1133.312,A 0.000,B 0.000,C 90.000,E1 92.178} C_DIS
LIN {X -0.062,Y -562.575,Z 1133.306,A 0.000,B 0.000,C 90.000,E1 91.088} C_DIS
LIN {X -0.005,Y -563.668,Z 1133.297,A 0.000,B 0.000,C 90.000,E1 89.427} C_DIS
LIN {X -0.145,Y -564.260,Z 1133.291,A 0.000,B 0.000,C 90.000,E1 88.339} C_DIS
LIN {X -0.017,Y -565.217,Z 1133.282,A 0.000,B 0.000,C 90.000,E1 86.674} C_DIS
LIN {X -0.011,Y -565.929,Z 1133.274,A 0.000,B 0.000,C 90.000,E1 85.298} C_DIS
LIN {X 0.202,Y -566.618,Z 1133.265,A 0.000,B 0.000,C 90.000,E1 83.628} C_DIS
LIN {X -0.061,Y -567.400,Z 1133.256,A 0.000,B 0.000,C 90.000,E1 82.008} C_DIS
LIN {X 0.253,Y -568.113,Z 1133.246,A 0.000,B 0.000,C 90.000,E1 80.330} C_DIS
LIN {X 0.109,Y -568.815,Z 1133.237,A 0.000,B 0.000,C 90.000,E1 78.701} C_DIS
LIN {X 0.086,Y -569.621,Z 1133.228,A 0.000,B 0.000,C 90.000,E1 77.061} C_DIS
LIN {X 0.210,Y -570.363,Z 1133.219,A 0.000,B 0.000,C 90.000,E1 75.408} C_DIS
LIN {X -0.046,Y -571.339,Z 1133.210,A 0.000,B 0.000,C 90.000,E1 73.795} C_DIS
LIN {X -0.277,Y -572.394,Z 1133.201,A 0.000,B 0.000,C 90.000,E1 72.181} C_DIS
LIN {X -0.316,Y -573.637,Z 1133.192,A 0.000,B 0.000,C 90.000,E1 70.550} C_DIS
LIN {X -0.138,Y -575.054,Z 1133.183,A 0.000,B 0.000,C 90.000,E1 68.901} C_DIS
LIN {X 0.126,Y -576.888,Z 1133.172,A 0.000,B 0.000,C 90.000,E1 66.975} C_DIS
LIN {X -0.094,Y -578.520,Z 1133.162,A 0.000,B 0.000,C 90.000,E1 65.101} C_DIS
LIN {X -0.002,Y -579.241,Z 1133.157,A 0.000,B 0.000,C 90.000,E1 64.280} C_DIS
LIN {X 0.078,Y -580.407,Z 1133.150,A 0.000,B 0.000,C 90.000,E1 62.922} C_DIS
LIN {X 0.050,Y -581.740,Z 1133.141,A 0.000,B 0.000,C 90.000,E1 61.307} C_DIS
LIN {X 0.324,Y -582.884,Z 1133.132,A 0.000,B 0.000,C 90.000,E1 59.665} C_DIS
LIN {X 0.247,Y -583.779,Z 1133.124,A 0.000,B 0.000,C 90.000,E1 58.329} C_DIS
LIN {X -0.314,Y -584.566,Z 1133.117,A 0.000,B 0.000,C 90.000,E1 57.041} C_DIS
LIN {X 0.129,Y -585.483,Z 1133.108,A 0.000,B 0.000,C 90.000,E1 55.388} C_DIS
LIN {X -0.177,Y -586.509,Z 1133.097,A 0.000,B 0.000,C 90.000,E1 53.543} C_DIS
LIN {X 0.048,Y -586.907,Z 1133.093,A 0.000,B 0.000,C 90.000,E1 52.718} C_DIS
LIN {X 0.027,Y -587.722,Z 1133.083,A 0.000,B 0.000,C 90.000,E1 50.848} C_DIS
LIN {X -0.025,Y -588.003,Z 1133.077,A 0.000,B 0.000,C 90.000,E1 49.784} C_DIS
LIN {X 0.233,Y -588.133,Z 1133.071,A 0.000,B 0.000,C 90.000,E1 48.690} C_DIS
LIN {X 0.041,Y -587.988,Z 1133.062,A 0.000,B 0.000,C 90.000,E1 47.106} C_DIS
LIN {X -0.124,Y -587.767,Z 1133.056,A 0.000,B 0.000,C 90.000,E1 46.053} C_DIS
LIN {X -0.284,Y -587.406,Z 1133.050,A 0.000,B 0.000,C 90.000,E1 45.000} C_DIS
LIN {X -0.199,Y -587.035,Z 1133.045,A 0.000,B 0.000,C 90.000,E1 44.190} C_DIS
LIN {X -0.197,Y -586.238,Z 1133.038,A 0.000,B 0.000,C 90.000,E1 42.852} C_DIS
LIN {X 0.122,Y -585.659,Z 1133.035,A 0.000,B 0.000,C 90.000,E1 42.285} C_DIS
LIN {X -0.135,Y -585.499,Z 1133.034,A 0.000,B 0.000,C 90.000,E1 42.043} C_DIS
LIN {X 0.057,Y -583.624,Z 1133.025,A 0.000,B 0.000,C 90.000,E1 40.415} C_DIS
LIN {X -0.032,Y -583.019,Z 1133.022,A 0.000,B 0.000,C 90.000,E1 39.886} C_DIS
LIN {X -0.054,Y -581.058,Z 1133.014,A 0.000,B 0.000,C 90.000,E1 38.543} C_DIS
LIN {X 0.337,Y -578.660,Z 1133.007,A 0.000,B 0.000,C 90.000,E1 37.156} C_DIS
LIN {X 0.016,Y -576.924,Z 1133.002,A 0.000,B 0.000,C 90.000,E1 36.377} C_DIS
LIN {X -0.319,Y -574.927,Z 1132.998,A 0.000,B 0.000,C 90.000,E1 35.598} C_DIS
LIN {X -0.021,Y -573.446,Z 1132.995,A 0.000,B 0.000,C 90.000,E1 35.025} C_DIS
LIN {X 0.209,Y -569.992,Z 1132.989,A 0.000,B 0.000,C 90.000,E1 33.913} C_DIS
LIN {X 0.147,Y -567.995,Z 1132.985,A 0.000,B 0.000,C 90.000,E1 33.372} C_DIS
LIN {X 0.187,Y -564.782,Z 1132.981,A 0.000,B 0.000,C 90.000,E1 32.546} C_DIS
LIN {X -0.009,Y -561.819,Z 1132.977,A 0.000,B 0.000,C 90.000,E1 31.878} C_DIS
LIN {X -0.261,Y -556.476,Z 1132.971,A 0.000,B 0.000,C 90.000,E1 30.797} C_DIS
LIN {X -0.231,Y -549.633,Z 1132.964,A 0.000,B 0.000,C 90.000,E1 29.539} C_DIS
LIN {X 0.040,Y -546.335,Z 1132.961,A 0.000,B 0.000,C 90.000,E1 28.949} C_DIS
LIN {X -0.099,Y -540.061,Z 1132.955,A 0.000,B 0.000,C 90.000,E1 27.975} C_DIS
LIN {X -0.037,Y -534.982,Z 1132.951,A 0.000,B 0.000,C 90.000,E1 27.257} C_DIS
LIN {X -0.173,Y -528.523,Z 1132.947,A 0.000,B 0.000,C 90.000,E1 26.411} C_DIS
LIN {X 0.017,Y -522.677,Z 1132.943,A 0.000,B 0.000,C 90.000,E1 25.668} C_DIS
LIN {X -0.153,Y -515.113,Z 1132.938,A 0.000,B 0.000,C 90.000,E1 24.823} C_DIS
LIN {X 0.059,Y -508.470,Z 1132.934,A 0.000,B 0.000,C 90.000,E1 24.079} C_DIS
LIN {X 0.056,Y -500.527,Z 1132.929,A 0.000,B 0.000,C 90.000,E1 23.259} C_DIS
LIN {X 0.000,Y -492.283,Z 1132.925,A 0.000,B 0.000,C 90.000,E1 22.461} C_DIS
LIN {X 0.190,Y -486.524,Z 1132.922,A 0.000,B 0.000,C 90.000,E1 21.897} C_DIS
LIN {X -0.206,Y -479.290,Z 1132.918,A 0.000,B 0.000,C 90.000,E1 21.280} C_DIS
LIN {X 0.034,Y -469.211,Z 1132.913,A 0.000,B 0.000,C 90.000,E1 20.355} C_DIS
LIN {X 0.169,Y -453.135,Z 1132.905,A 0.000,B 0.000,C 90.000,E1 18.906} C_DIS
LIN {X -0.131,Y -437.244,Z 1132.897,A 0.000,B 0.000,C 90.000,E1 17.457} C_DIS
LIN {X 0.001,Y -423.077,Z 1132.889,A 0.000,B 0.000,C 90.000,E1 15.969} C_DIS
LIN {X 0.003,Y -412.131,Z 1132.882,A 0.000,B 0.000,C 90.000,E1 14.717} C_DIS
LIN {X 0.015,Y -404.187,Z 1132.876,A 0.000,B 0.000,C 90.000,E1 13.703} C_DIS
LIN {X 0.058,Y -400.480,Z 1132.873,A 0.000,B 0.000,C 90.000,E1 13.175} C_DIS
LIN {X 0.082,Y -397.214,Z 1132.870,A 0.000,B 0.000,C 90.000,E1 12.647} C_DIS
LIN {X 0.131,Y -394.201,Z 1132.867,A 0.000,B 0.000,C 90.000,E1 12.063} C_DIS
LIN {X -0.127,Y -392.706,Z 1132.865,A 0.000,B 0.000,C 90.000,E1 11.658} C_DIS
LIN {X 0.088,Y -392.110,Z 1132.861,A 0.000,B 0.000,C 90.000,E1 11.007} C_DIS
LIN {X 0.180,Y -392.671,Z 1132.858,A 0.000,B 0.000,C 90.000,E1 10.366} C_DIS
LIN {X 0.036,Y -394.178,Z 1132.854,A 0.000,B 0.000,C 90.000,E1 9.613} C_DIS
LIN {X -0.105,Y -397.963,Z 1132.846,A 0.000,B 0.000,C 90.000,E1 8.219} C_DIS
LIN {X 0.143,Y -403.326,Z 1132.836,A 0.000,B 0.000,C 90.000,E1 6.429} C_DIS
LIN {X 0.112,Y -405.294,Z 1132.833,A 0.000,B 0.000,C 90.000,E1 5.910} C_DIS
LIN {X -0.176,Y -407.762,Z 1132.830,A 0.000,B 0.000,C 90.000,E1 5.448} C_DIS
LIN {X -0.207,Y -411.826,Z 1132.827,A 0.000,B 0.000,C 90.000,E1 4.935} C_DIS
LIN {X 0.111,Y -415.343,Z 1132.826,A 0.000,B 0.000,C 90.000,E1 4.588} C_DIS
LIN {X -0.023,Y -416.943,Z 1132.825,A 0.000,B 0.000,C 90.000,E1 4.473} C_DIS
LIN {X -0.144,Y -424.541,Z 1132.822,A 0.000,B 0.000,C 90.000,E1 3.955} C_DIS
LIN {X -0.096,Y -445.747,Z 1132.814,A 0.000,B 0.000,C 90.000,E1 2.465} C_DIS
LIN {X 0.039,Y -461.841,Z 1132.808,A 0.000,B 0.000,C 90.000,E1 1.375} C_DIS
LIN {X 0.120,Y -474.805,Z 1132.803,A 0.000,B 0.000,C 90.000,E1 0.516} C_DIS
LIN {X 0.000,Y -482.697,Z 1132.800,A 0.000,B 0.000,C 90.000,E1 360.000} C_DIS
LIN {X -0.233,Y -490.361,Z 1132.797,A 0.000,B 0.000,C 90.000,E1 359.484} C_DIS
LIN {X -0.230,Y -497.940,Z 1132.794,A 0.000,B 0.000,C 90.000,E1 358.912} C_DIS
LIN {X 0.079,Y -503.971,Z 1132.791,A 0.000,B 0.000,C 90.000,E1 358.396} C_DIS
LIN {X 0.129,Y -511.170,Z 1132.788,A 0.000,B 0.000,C 90.000,E1 357.764} C_DIS
LIN {X 0.229,Y -516.683,Z 1132.785,A 0.000,B 0.000,C 90.000,E1 357.249} C_DIS
LIN {X 0.036,Y -521.992,Z 1132.782,A 0.000,B 0.000,C 90.000,E1 356.731} C_DIS
LIN {X 0.231,Y -528.067,Z 1132.778,A 0.000,B 0.000,C 90.000,E1 356.045} C_DIS
LIN {X 0.216,Y -532.913,Z 1132.775,A 0.000,B 0.000,C 90.000,E1 355.469} C_DIS
LIN {X 0.231,Y -537.352,Z 1132.772,A 0.000,B 0.000,C 90.000,E1 354.894} C_DIS
LIN {X 0.014,Y -542.294,Z 1132.768,A 0.000,B 0.000,C 90.000,E1 354.204} C_DIS
LIN {X -0.167,Y -546.730,Z 1132.764,A 0.000,B 0.000,C 90.000,E1 353.514} C_DIS
LIN {X -0.246,Y -550.755,Z 1132.760,A 0.000,B 0.000,C 90.000,E1 352.818} C_DIS
LIN {X 0.266,Y -554.399,Z 1132.756,A 0.000,B 0.000,C 90.000,E1 352.064} C_DIS
LIN {X 0.138,Y -556.464,Z 1132.754,A 0.000,B 0.000,C 90.000,E1 351.659} C_DIS
LIN {X 0.070,Y -559.490,Z 1132.750,A 0.000,B 0.000,C 90.000,E1 350.971} C_DIS
LIN {X -0.048,Y -562.812,Z 1132.745,A 0.000,B 0.000,C 90.000,E1 350.151} C_DIS
LIN {X -0.061,Y -566.743,Z 1132.739,A 0.000,B 0.000,C 90.000,E1 349.050} C_DIS
LIN {X 0.087,Y -570.334,Z 1132.733,A 0.000,B 0.000,C 90.000,E1 347.937} C_DIS
LIN {X -0.078,Y -574.408,Z 1132.725,A 0.000,B 0.000,C 90.000,E1 346.589} C_DIS
LIN {X -0.248,Y -577.389,Z 1132.719,A 0.000,B 0.000,C 90.000,E1 345.519} C_DIS
LIN {X 0.189,Y -580.311,Z 1132.714,A 0.000,B 0.000,C 90.000,E1 344.393} C_DIS
LIN {X 0.106,Y -583.076,Z 1132.707,A 0.000,B 0.000,C 90.000,E1 343.323} C_DIS
LIN {X -0.100,Y -586.405,Z 1132.700,A 0.000,B 0.000,C 90.000,E1 342.000} C_DIS
LIN {X 0.072,Y -588.812,Z 1132.694,A 0.000,B 0.000,C 90.000,E1 340.913} C_DIS
LIN {X 0.044,Y -590.516,Z 1132.690,A 0.000,B 0.000,C 90.000,E1 340.115} C_DIS
LIN {X 0.157,Y -593.088,Z 1132.682,A 0.000,B 0.000,C 90.000,E1 338.773} C_DIS
LIN {X 0.176,Y -594.510,Z 1132.678,A 0.000,B 0.000,C 90.000,E1 337.975} C_DIS
LIN {X 0.205,Y -595.606,Z 1132.673,A 0.000,B 0.000,C 90.000,E1 337.177} C_DIS
LIN {X 0.148,Y -596.853,Z 1132.667,A 0.000,B 0.000,C 90.000,E1 336.125} C_DIS
LIN {X -0.276,Y -597.876,Z 1132.660,A 0.000,B 0.000,C 90.000,E1 334.845} C_DIS
LIN {X 0.024,Y -598.236,Z 1132.656,A 0.000,B 0.000,C 90.000,E1 334.024} C_DIS
LIN {X -0.133,Y -598.259,Z 1132.653,A 0.000,B 0.000,C 90.000,E1 333.512} C_DIS
LIN {X 0.082,Y -597.878,Z 1132.647,A 0.000,B 0.000,C 90.000,E1 332.436} C_DIS
LIN {X 0.120,Y -597.254,Z 1132.643,A 0.000,B 0.000,C 90.000,E1 331.641} C_DIS
LIN {X -0.047,Y -596.678,Z 1132.640,A 0.000,B 0.000,C 90.000,E1 331.129} C_DIS
LIN {X 0.071,Y -595.970,Z 1132.637,A 0.000,B 0.000,C 90.000,E1 330.589} C_DIS
LIN {X 0.098,Y -594.481,Z 1132.632,A 0.000,B 0.000,C 90.000,E1 329.793} C_DIS
LIN {X -0.094,Y -593.302,Z 1132.629,A 0.000,B 0.000,C 90.000,E1 329.282} C_DIS
LIN {X 0.209,Y -591.050,Z 1132.625,A 0.000,B 0.000,C 90.000,E1 328.456} C_DIS
LIN {X 0.180,Y -588.265,Z 1132.620,A 0.000,B 0.000,C 90.000,E1 327.661} C_DIS
LIN {X -0.056,Y -584.883,Z 1132.616,A 0.000,B 0.000,C 90.000,E1 326.882} C_DIS
LIN {X -0.011,Y -582.354,Z 1132.613,A 0.000,B 0.000,C 90.000,E1 326.342} C_DIS
LIN {X 0.178,Y -577.974,Z 1132.609,A 0.000,B 0.000,C 90.000,E1 325.515} C_DIS
LIN {X 0.073,Y -573.944,Z 1132.605,A 0.000,B 0.000,C 90.000,E1 324.848} C_DIS
LIN {X -0.341,Y -571.406,Z 1132.603,A 0.000,B 0.000,C 90.000,E1 324.482} C_DIS
LIN {X -0.070,Y -567.703,Z 1132.599,A 0.000,B 0.000,C 90.000,E1 323.909} C_DIS
LIN {X 0.059,Y -562.604,Z 1132.596,A 0.000,B 0.000,C 90.000,E1 323.210} C_DIS
LIN {X -0.183,Y -558.233,Z 1132.593,A 0.000,B 0.000,C 90.000,E1 322.683} C_DIS
LIN {X -0.155,Y -554.884,Z 1132.590,A 0.000,B 0.000,C 90.000,E1 322.271} C_DIS
LIN {X 0.036,Y -542.965,Z 1132.583,A 0.000,B 0.000,C 90.000,E1 320.884} C_DIS
LIN {X 0.061,Y -535.648,Z 1132.578,A 0.000,B 0.000,C 90.000,E1 320.033} C_DIS
LIN {X 0.058,Y -532.358,Z 1132.575,A 0.000,B 0.000,C 90.000,E1 319.542} C_DIS
LIN {X 0.227,Y -531.493,Z 1132.574,A 0.000,B 0.000,C 90.000,E1 319.380} C_DIS
LIN {X -0.023,Y -529.319,Z 1132.572,A 0.000,B 0.000,C 90.000,E1 318.976} C_DIS
LIN {X 0.085,Y -526.689,Z 1132.568,A 0.000,B 0.000,C 90.000,E1 318.243} C_DIS
LIN {X -0.186,Y -525.698,Z 1132.566,A 0.000,B 0.000,C 90.000,E1 317.838} C_DIS
LIN {X -0.029,Y -525.274,Z 1132.565,A 0.000,B 0.000,C 90.000,E1 317.676} C_DIS
LIN {X 0.125,Y -524.261,Z 1132.560,A 0.000,B 0.000,C 90.000,E1 316.743} C_DIS
LIN {X -0.186,Y -524.017,Z 1132.552,A 0.000,B 0.000,C 90.000,E1 315.324} C_DIS
LIN {X 0.168,Y -524.161,Z 1132.542,A 0.000,B 0.000,C 90.000,E1 313.542} C_DIS
LIN {X -0.159,Y -525.289,Z 1132.523,A 0.000,B 0.000,C 90.000,E1 310.092} C_DIS
LIN {X 0.261,Y -526.424,Z 1132.511,A 0.000,B 0.000,C 90.000,E1 308.016} C_DIS
LIN {X 0.088,Y -527.538,Z 1132.502,A 0.000,B 0.000,C 90.000,E1 306.297} C_DIS
LIN {X 0.018,Y -529.111,Z 1132.489,A 0.000,B 0.000,C 90.000,E1 303.992} C_DIS
LIN {X 0.048,Y -530.103,Z 1132.481,A 0.000,B 0.000,C 90.000,E1 302.546} C_DIS
LIN {X 0.238,Y -531.456,Z 1132.471,A 0.000,B 0.000,C 90.000,E1 300.797} C_DIS
LIN {X -0.247,Y -532.508,Z 1132.463,A 0.000,B 0.000,C 90.000,E1 299.411} C_DIS
LIN {X -0.248,Y -533.441,Z 1132.455,A 0.000,B 0.000,C 90.000,E1 297.975} C_DIS
LIN {X 0.045,Y -533.971,Z 1132.449,A 0.000,B 0.000,C 90.000,E1 296.796} C_DIS
LIN {X -0.133,Y -534.311,Z 1132.443,A 0.000,B 0.000,C 90.000,E1 295.668} C_DIS
LIN {X -0.073,Y -534.433,Z 1132.436,A 0.000,B 0.000,C 90.000,E1 294.515} C_DIS
LIN {X -0.035,Y -534.467,Z 1132.428,A 0.000,B 0.000,C 90.000,E1 293.078} C_DIS
LIN {X -0.002,Y -534.458,Z 1132.420,A 0.000,B 0.000,C 90.000,E1 291.642} C_DIS
LIN {X 0.143,Y -534.352,Z 1132.412,A 0.000,B 0.000,C 90.000,E1 290.194} C_DIS
LIN {X -0.001,Y -534.070,Z 1132.403,A 0.000,B 0.000,C 90.000,E1 288.489} C_DIS
LIN {X -0.323,Y -533.583,Z 1132.393,A 0.000,B 0.000,C 90.000,E1 286.804} C_DIS
LIN {X 0.133,Y -533.119,Z 1132.387,A 0.000,B 0.000,C 90.000,E1 285.607} C_DIS
LIN {X -0.076,Y -532.592,Z 1132.380,A 0.000,B 0.000,C 90.000,E1 284.481} C_DIS
LIN {X -0.253,Y -531.890,Z 1132.372,A 0.000,B 0.000,C 90.000,E1 283.063} C_DIS
LIN {X 0.108,Y -530.967,Z 1132.363,A 0.000,B 0.000,C 90.000,E1 281.299} C_DIS
LIN {X 0.202,Y -530.111,Z 1132.355,A 0.000,B 0.000,C 90.000,E1 279.849} C_DIS
LIN {X -0.204,Y -529.207,Z 1132.345,A 0.000,B 0.000,C 90.000,E1 278.163} C_DIS
LIN {X -0.227,Y -528.167,Z 1132.334,A 0.000,B 0.000,C 90.000,E1 276.144} C_DIS
LIN {X 0.237,Y -527.422,Z 1132.324,A 0.000,B 0.000,C 90.000,E1 274.359} C_DIS
LIN {X 0.144,Y -526.798,Z 1132.316,A 0.000,B 0.000,C 90.000,E1 272.922} C_DIS
LIN {X -0.024,Y -526.041,Z 1132.307,A 0.000,B 0.000,C 90.000,E1 271.203} C_DIS
LIN {X -0.184,Y -525.378,Z 1132.299,A 0.000,B 0.000,C 90.000,E1 269.771} C_DIS
LIN {X 0.168,Y -524.732,Z 1132.291,A 0.000,B 0.000,C 90.000,E1 268.282} C_DIS
LIN {X -0.021,Y -523.814,Z 1132.281,A 0.000,B 0.000,C 90.000,E1 266.560} C_DIS
LIN {X -0.223,Y -522.838,Z 1132.271,A 0.000,B 0.000,C 90.000,E1 264.837} C_DIS
LIN {X 0.176,Y -521.951,Z 1132.265,A 0.000,B 0.000,C 90.000,E1 263.628} C_DIS
LIN {X 0.027,Y -519.967,Z 1132.253,A 0.000,B 0.000,C 90.000,E1 261.602} C_DIS
LIN {X -0.077,Y -518.203,Z 1132.244,A 0.000,B 0.000,C 90.000,E1 259.859} C_DIS
LIN {X -0.125,Y -516.523,Z 1132.234,A 0.000,B 0.000,C 90.000,E1 258.105} C_DIS
LIN {X -0.219,Y -514.759,Z 1132.224,A 0.000,B 0.000,C 90.000,E1 256.353} C_DIS
LIN {X -0.117,Y -513.197,Z 1132.214,A 0.000,B 0.000,C 90.000,E1 254.574} C_DIS
LIN {X -0.015,Y -511.785,Z 1132.206,A 0.000,B 0.000,C 90.000,E1 253.087} C_DIS
LIN {X 0.206,Y -510.286,Z 1132.198,A 0.000,B 0.000,C 90.000,E1 251.583} C_DIS
LIN {X 0.085,Y -508.700,Z 1132.190,A 0.000,B 0.000,C 90.000,E1 250.115} C_DIS
LIN {X -0.057,Y -507.020,Z 1132.181,A 0.000,B 0.000,C 90.000,E1 248.646} C_DIS
LIN {X 0.136,Y -505.686,Z 1132.175,A 0.000,B 0.000,C 90.000,E1 247.433} C_DIS
LIN {X 0.229,Y -504.231,Z 1132.168,A 0.000,B 0.000,C 90.000,E1 246.230} C_DIS
LIN {X 0.098,Y -502.707,Z 1132.161,A 0.000,B 0.000,C 90.000,E1 245.049} C_DIS
LIN {X -0.011,Y -500.562,Z 1132.153,A 0.000,B 0.000,C 90.000,E1 243.563} C_DIS
LIN {X 0.295,Y -498.353,Z 1132.145,A 0.000,B 0.000,C 90.000,E1 242.025} C_DIS
LIN {X -0.048,Y -495.534,Z 1132.135,A 0.000,B 0.000,C 90.000,E1 240.255} C_DIS
LIN {X -0.048,Y -492.999,Z 1132.126,A 0.000,B 0.000,C 90.000,E1 238.742} C_DIS
LIN {X -0.263,Y -490.510,Z 1132.118,A 0.000,B 0.000,C 90.000,E1 237.248} C_DIS
LIN {X -0.013,Y -487.468,Z 1132.108,A 0.000,B 0.000,C 90.000,E1 235.388} C_DIS
LIN {X -0.067,Y -484.901,Z 1132.099,A 0.000,B 0.000,C 90.000,E1 233.863} C_DIS
LIN {X 0.030,Y -481.155,Z 1132.087,A 0.000,B 0.000,C 90.000,E1 231.698} C_DIS
LIN {X 0.244,Y -478.961,Z 1132.080,A 0.000,B 0.000,C 90.000,E1 230.436} C_DIS
LIN {X -0.042,Y -475.538,Z 1132.070,A 0.000,B 0.000,C 90.000,E1 228.609} C_DIS
LIN {X -0.273,Y -473.367,Z 1132.063,A 0.000,B 0.000,C 90.000,E1 227.391} C_DIS
LIN {X 0.044,Y -469.542,Z 1132.051,A 0.000,B 0.000,C 90.000,E1 225.162} C_DIS
LIN {X 0.078,Y -465.210,Z 1132.035,A 0.000,B 0.000,C 90.000,E1 222.324} C_DIS
LIN {X -0.051,Y -461.727,Z 1132.021,A 0.000,B 0.000,C 90.000,E1 219.806} C_DIS
LIN {X 0.022,Y -459.056,Z 1132.009,A 0.000,B 0.000,C 90.000,E1 217.569} C_DIS
LIN {X 0.084,Y -457.002,Z 1131.998,A 0.000,B 0.000,C 90.000,E1 215.644} C_DIS
LIN {X -0.056,Y -453.651,Z 1131.979,A 0.000,B 0.000,C 90.000,E1 212.133} C_DIS
LIN {X -0.195,Y -452.566,Z 1131.970,A 0.000,B 0.000,C 90.000,E1 210.541} C_DIS
LIN {X 0.145,Y -451.534,Z 1131.950,A 0.000,B 0.000,C 90.000,E1 206.950} C_DIS
LIN {X 0.148,Y -452.024,Z 1131.941,A 0.000,B 0.000,C 90.000,E1 205.335} C_DIS
LIN {X -0.228,Y -453.349,Z 1131.932,A 0.000,B 0.000,C 90.000,E1 203.770} C_DIS
LIN {X -0.156,Y -455.797,Z 1131.923,A 0.000,B 0.000,C 90.000,E1 202.153} C_DIS
LIN {X -0.204,Y -458.934,Z 1131.914,A 0.000,B 0.000,C 90.000,E1 200.556} C_DIS
LIN {X 0.166,Y -463.619,Z 1131.903,A 0.000,B 0.000,C 90.000,E1 198.598} C_DIS
LIN {X 0.101,Y -471.448,Z 1131.889,A 0.000,B 0.000,C 90.000,E1 196.079} C_DIS
LIN {X -0.238,Y -477.965,Z 1131.879,A 0.000,B 0.000,C 90.000,E1 194.245} C_DIS
LIN {X 0.129,Y -488.294,Z 1131.864,A 0.000,B 0.000,C 90.000,E1 191.422} C_DIS
LIN {X -0.058,Y -498.508,Z 1131.849,A 0.000,B 0.000,C 90.000,E1 188.859} C_DIS
LIN {X 0.165,Y -505.197,Z 1131.840,A 0.000,B 0.000,C 90.000,E1 187.182} C_DIS
LIN {X -0.245,Y -511.114,Z 1131.832,A 0.000,B 0.000,C 90.000,E1 185.739} C_DIS
LIN {X -0.089,Y -517.023,Z 1131.824,A 0.000,B 0.000,C 90.000,E1 184.245} C_DIS
LIN {X 0.135,Y -524.214,Z 1131.814,A 0.000,B 0.000,C 90.000,E1 182.465} C_DIS
LIN {X 0.235,Y -530.681,Z 1131.805,A 0.000,B 0.000,C 90.000,E1 180.859} C_DIS
LIN {X -0.074,Y -538.356,Z 1131.795,A 0.000,B 0.000,C 90.000,E1 179.026} C_DIS
LIN {X 0.007,Y -543.104,Z 1131.788,A 0.000,B 0.000,C 90.000,E1 177.879} C_DIS
LIN {X 0.081,Y -551.984,Z 1131.776,A 0.000,B 0.000,C 90.000,E1 175.755} C_DIS
LIN {X 0.230,Y -558.475,Z 1131.768,A 0.000,B 0.000,C 90.000,E1 174.204} C_DIS
LIN {X -0.239,Y -565.494,Z 1131.759,A 0.000,B 0.000,C 90.000,E1 172.591} C_DIS
LIN {X -0.211,Y -570.232,Z 1131.753,A 0.000,B 0.000,C 90.000,E1 171.489} C_DIS
LIN {X 0.087,Y -576.032,Z 1131.745,A 0.000,B 0.000,C 90.000,E1 170.095} C_DIS
LIN {X 0.046,Y -579.422,Z 1131.741,A 0.000,B 0.000,C 90.000,E1 169.285} C_DIS
LIN {X 0.042,Y -584.893,Z 1131.733,A 0.000,B 0.000,C 90.000,E1 167.937} C_DIS
LIN {X 0.135,Y -590.205,Z 1131.726,A 0.000,B 0.000,C 90.000,E1 166.589} C_DIS
LIN {X 0.189,Y -594.289,Z 1131.720,A 0.000,B 0.000,C 90.000,E1 165.519} C_DIS
LIN {X 0.146,Y -598.172,Z 1131.714,A 0.000,B 0.000,C 90.000,E1 164.464} C_DIS
LIN {X -0.099,Y -601.791,Z 1131.708,A 0.000,B 0.000,C 90.000,E1 163.433} C_DIS
LIN {X 0.333,Y -606.935,Z 1131.699,A 0.000,B 0.000,C 90.000,E1 161.819} C_DIS
LIN {X -0.038,Y -610.917,Z 1131.692,A 0.000,B 0.000,C 90.000,E1 160.550} C_DIS
LIN {X -0.095,Y -613.989,Z 1131.686,A 0.000,B 0.000,C 90.000,E1 159.518} C_DIS
LIN {X -0.149,Y -617.527,Z 1131.679,A 0.000,B 0.000,C 90.000,E1 158.230} C_DIS
LIN {X 0.080,Y -621.629,Z 1131.670,A 0.000,B 0.000,C 90.000,E1 156.666} C_DIS
LIN {X -0.174,Y -624.904,Z 1131.663,A 0.000,B 0.000,C 90.000,E1 155.409} C_DIS
LIN {X 0.186,Y -628.062,Z 1131.656,A 0.000,B 0.000,C 90.000,E1 154.101} C_DIS
LIN {X -0.264,Y -631.051,Z 1131.649,A 0.000,B 0.000,C 90.000,E1 152.871} C_DIS
LIN {X -0.138,Y -633.322,Z 1131.644,A 0.000,B 0.000,C 90.000,E1 151.847} C_DIS
LIN {X -0.195,Y -636.078,Z 1131.637,A 0.000,B 0.000,C 90.000,E1 150.589} C_DIS
LIN {X -0.199,Y -638.711,Z 1131.630,A 0.000,B 0.000,C 90.000,E1 149.331} C_DIS
LIN {X -0.167,Y -641.234,Z 1131.623,A 0.000,B 0.000,C 90.000,E1 148.074} C_DIS
LIN {X 0.107,Y -644.036,Z 1131.614,A 0.000,B 0.000,C 90.000,E1 146.548} C_DIS
LIN {X 0.082,Y -646.694,Z 1131.606,A 0.000,B 0.000,C 90.000,E1 145.055} C_DIS
LIN {X -0.065,Y -649.211,Z 1131.598,A 0.000,B 0.000,C 90.000,E1 143.577} C_DIS
LIN {X 0.224,Y -651.720,Z 1131.589,A 0.000,B 0.000,C 90.000,E1 142.065} C_DIS
LIN {X -0.055,Y -655.268,Z 1131.578,A 0.000,B 0.000,C 90.000,E1 140.114} C_DIS
LIN {X 0.306,Y -657.611,Z 1131.572,A 0.000,B 0.000,C 90.000,E1 138.852} C_DIS
LIN {X 0.178,Y -660.512,Z 1131.563,A 0.000,B 0.000,C 90.000,E1 137.391} C_DIS
LIN {X 0.069,Y -664.451,Z 1131.553,A 0.000,B 0.000,C 90.000,E1 135.445} C_DIS
LIN {X 0.068,Y -669.349,Z 1131.540,A 0.000,B 0.000,C 90.000,E1 133.257} C_DIS
LIN {X -0.308,Y -673.404,Z 1131.531,A 0.000,B 0.000,C 90.000,E1 131.595} C_DIS
LIN {X -0.156,Y -676.299,Z 1131.524,A 0.000,B 0.000,C 90.000,E1 130.378} C_DIS
LIN {X -0.046,Y -682.362,Z 1131.511,A 0.000,B 0.000,C 90.000,E1 127.971} C_DIS
LIN {X 0.195,Y -684.750,Z 1131.506,A 0.000,B 0.000,C 90.000,E1 126.996} C_DIS
LIN {X 0.224,Y -687.768,Z 1131.499,A 0.000,B 0.000,C 90.000,E1 125.804} C_DIS
LIN {X 0.308,Y -690.681,Z 1131.492,A 0.000,B 0.000,C 90.000,E1 124.612} C_DIS
LIN {X 0.078,Y -694.149,Z 1131.485,A 0.000,B 0.000,C 90.000,E1 123.214} C_DIS
LIN {X -0.157,Y -696.330,Z 1131.479,A 0.000,B 0.000,C 90.000,E1 122.291} C_DIS
LIN {X 0.014,Y -698.297,Z 1131.474,A 0.000,B 0.000,C 90.000,E1 121.337} C_DIS
LIN {X 0.202,Y -700.000,Z 1131.469,A 0.000,B 0.000,C 90.000,E1 120.384} C_DIS
LIN {X 0.257,Y -702.855,Z 1131.460,A 0.000,B 0.000,C 90.000,E1 118.743} C_DIS
LIN {X 0.146,Y -704.032,Z 1131.456,A 0.000,B 0.000,C 90.000,E1 118.052} C_DIS
LIN {X -0.244,Y -704.926,Z 1131.452,A 0.000,B 0.000,C 90.000,E1 117.385} C_DIS
LIN {X -0.008,Y -705.546,Z 1131.448,A 0.000,B 0.000,C 90.000,E1 116.668} C_DIS
LIN {X 0.210,Y -706.120,Z 1131.443,A 0.000,B 0.000,C 90.000,E1 115.720} C_DIS
LIN {X 0.147,Y -706.284,Z 1131.439,A 0.000,B 0.000,C 90.000,E1 115.027} C_DIS
LIN {X -0.205,Y -706.157,Z 1131.437,A 0.000,B 0.000,C 90.000,E1 114.591} C_DIS
LIN {X 0.378,Y -705.338,Z 1131.434,A 0.000,B 0.000,C 90.000,E1 114.079} C_DIS
LIN {X -0.265,Y -704.811,Z 1131.433,A 0.000,B 0.000,C 90.000,E1 113.898} C_DIS
LIN {X 0.305,Y -702.871,Z 1131.430,A 0.000,B 0.000,C 90.000,E1 113.387} C_DIS
LIN {X 0.166,Y -702.300,Z 1131.429,A 0.000,B 0.000,C 90.000,E1 113.281} C_DIS
LIN {X -0.339,Y -701.434,Z 1131.429,A 0.000,B 0.000,C 90.000,E1 113.206} C_DIS
LIN {X -0.070,Y -697.049,Z 1131.426,A 0.000,B 0.000,C 90.000,E1 112.717} C_DIS
LIN {X 0.059,Y -695.467,Z 1131.426,A 0.000,B 0.000,C 90.000,E1 112.589} C_DIS
LIN {X 0.187,Y -692.703,Z 1131.425,A 0.000,B 0.000,C 90.000,E1 112.461} C_DIS
LIN {X -0.039,Y -687.084,Z 1131.424,A 0.000,B 0.000,C 90.000,E1 112.280} C_DIS
LIN {X 0.133,Y -685.020,Z 1131.423,A 0.000,B 0.000,C 90.000,E1 112.206} C_DIS
LIN {X -0.270,Y -676.401,Z 1131.423,A 0.000,B 0.000,C 90.000,E1 112.153} C_DIS
LIN {X -0.279,Y -603.158,Z 1131.423,A 0.000,B 0.000,C 90.000,E1 112.153} C_DIS
LIN {X 0.284,Y -600.002,Z 1131.422,A 0.000,B 0.000,C 90.000,E1 111.897} C_DIS
LIN {X -0.146,Y -595.523,Z 1131.420,A 0.000,B 0.000,C 90.000,E1 111.589} C_DIS
LIN {X 0.115,Y -581.365,Z 1131.413,A 0.000,B 0.000,C 90.000,E1 110.301} C_DIS
LIN {X 0.076,Y -574.359,Z 1131.410,A 0.000,B 0.000,C 90.000,E1 109.704} C_DIS
LIN {X -0.142,Y -568.339,Z 1131.407,A 0.000,B 0.000,C 90.000,E1 109.268} C_DIS
LIN {X -0.181,Y -561.832,Z 1131.405,A 0.000,B 0.000,C 90.000,E1 108.852} C_DIS
LIN {X 0.306,Y -555.234,Z 1131.403,A 0.000,B 0.000,C 90.000,E1 108.417} C_DIS
LIN {X -0.177,Y -550.731,Z 1131.401,A 0.000,B 0.000,C 90.000,E1 108.127} C_DIS
LIN {X 0.214,Y -549.507,Z 1131.399,A 0.000,B 0.000,C 90.000,E1 107.873} C_DIS
LIN {X 0.172,Y -549.495,Z 1131.399,A 0.000,B 0.000,C 90.000,E1 107.873} C_DIS
LIN {X 0.155,Y -549.218,Z 1131.397,A 0.000,B 0.000,C 90.000,E1 107.511} C_DIS
LIN {X 0.242,Y -550.396,Z 1131.387,A 0.000,B 0.000,C 90.000,E1 105.607} C_DIS
LIN {X -0.089,Y -552.348,Z 1131.373,A 0.000,B 0.000,C 90.000,E1 103.119} C_DIS
LIN {X 0.219,Y -554.052,Z 1131.362,A 0.000,B 0.000,C 90.000,E1 101.130} C_DIS
LIN {X 0.306,Y -555.267,Z 1131.354,A 0.000,B 0.000,C 90.000,E1 99.726} C_DIS
LIN {X -0.189,Y -556.850,Z 1131.345,A 0.000,B 0.000,C 90.000,E1 98.106} C_DIS
LIN {X -0.100,Y -558.354,Z 1131.336,A 0.000,B 0.000,C 90.000,E1 96.429} C_DIS
LIN {X -0.175,Y -559.601,Z 1131.328,A 0.000,B 0.000,C 90.000,E1 95.049} C_DIS
LIN {X -0.226,Y -560.729,Z 1131.320,A 0.000,B 0.000,C 90.000,E1 93.669} C_DIS
LIN {X 0.268,Y -561.732,Z 1131.313,A 0.000,B 0.000,C 90.000,E1 92.236} C_DIS
LIN {X 0.219,Y -562.635,Z 1131.305,A 0.000,B 0.000,C 90.000,E1 90.859} C_DIS
LIN {X 0.174,Y -563.562,Z 1131.297,A 0.000,B 0.000,C 90.000,E1 89.484} C_DIS
LIN {X 0.157,Y -564.322,Z 1131.290,A 0.000,B 0.000,C 90.000,E1 88.108} C_DIS
LIN {X 0.266,Y -565.242,Z 1131.280,A 0.000,B 0.000,C 90.000,E1 86.445} C_DIS
LIN {X -0.248,Y -565.928,Z 1131.273,A 0.000,B 0.000,C 90.000,E1 85.122} C_DIS
LIN {X 0.074,Y -566.747,Z 1131.262,A 0.000,B 0.000,C 90.000,E1 83.166} C_DIS
LIN {X 0.204,Y -567.350,Z 1131.255,A 0.000,B 0.000,C 90.000,E1 81.781} C_DIS
LIN {X 0.045,Y -568.067,Z 1131.245,A 0.000,B 0.000,C 90.000,E1 80.151} C_DIS
LIN {X 0.268,Y -569.073,Z 1131.233,A 0.000,B 0.000,C 90.000,E1 77.937} C_DIS
LIN {X 0.070,Y -569.684,Z 1131.226,A 0.000,B 0.000,C 90.000,E1 76.589} C_DIS
LIN {X -0.022,Y -570.646,Z 1131.215,A 0.000,B 0.000,C 90.000,E1 74.685} C_DIS
LIN {X 0.310,Y -571.316,Z 1131.209,A 0.000,B 0.000,C 90.000,E1 73.559} C_DIS
LIN {X -0.115,Y -572.628,Z 1131.198,A 0.000,B 0.000,C 90.000,E1 71.692} C_DIS
LIN {X -0.146,Y -573.917,Z 1131.189,A 0.000,B 0.000,C 90.000,E1 70.061} C_DIS
LIN {X -0.332,Y -575.140,Z 1131.182,A 0.000,B 0.000,C 90.000,E1 68.720} C_DIS
LIN {X 0.086,Y -576.735,Z 1131.173,A 0.000,B 0.000,C 90.000,E1 67.050} C_DIS
LIN {X -0.148,Y -578.352,Z 1131.162,A 0.000,B 0.000,C 90.000,E1 65.177} C_DIS
LIN {X -0.092,Y -579.528,Z 1131.155,A 0.000,B 0.000,C 90.000,E1 63.819} C_DIS
LIN {X -0.268,Y -580.666,Z 1131.147,A 0.000,B 0.000,C 90.000,E1 62.487} C_DIS
LIN {X -0.029,Y -581.521,Z 1131.141,A 0.000,B 0.000,C 90.000,E1 61.385} C_DIS
LIN {X -0.136,Y -582.514,Z 1131.134,A 0.000,B 0.000,C 90.000,E1 60.049} C_DIS
LIN {X 0.148,Y -583.560,Z 1131.125,A 0.000,B 0.000,C 90.000,E1 58.408} C_DIS
LIN {X 0.212,Y -584.206,Z 1131.119,A 0.000,B 0.000,C 90.000,E1 57.327} C_DIS
LIN {X 0.159,Y -585.115,Z 1131.110,A 0.000,B 0.000,C 90.000,E1 55.722} C_DIS
LIN {X -0.245,Y -585.680,Z 1131.104,A 0.000,B 0.000,C 90.000,E1 54.689} C_DIS
LIN {X 0.080,Y -586.584,Z 1131.095,A 0.000,B 0.000,C 90.000,E1 53.050} C_DIS
LIN {X -0.045,Y -587.213,Z 1131.086,A 0.000,B 0.000,C 90.000,E1 51.457} C_DIS
LIN {X 0.081,Y -587.565,Z 1131.081,A 0.000,B 0.000,C 90.000,E1 50.642} C_DIS
LIN {X -0.046,Y -587.772,Z 1131.075,A 0.000,B 0.000,C 90.000,E1 49.585} C_DIS
LIN {X -0.169,Y -587.870,Z 1131.070,A 0.000,B 0.000,C 90.000,E1 48.528} C_DIS
LIN {X 0.036,Y -587.683,Z 1131.061,A 0.000,B 0.000,C 90.000,E1 46.905} C_DIS
LIN {X 0.050,Y -587.321,Z 1131.053,A 0.000,B 0.000,C 90.000,E1 45.567} C_DIS
LIN {X -0.365,Y -586.746,Z 1131.046,A 0.000,B 0.000,C 90.000,E1 44.271} C_DIS
LIN {X 0.031,Y -585.932,Z 1131.038,A 0.000,B 0.000,C 90.000,E1 42.894} C_DIS
LIN {X 0.046,Y -584.585,Z 1131.031,A 0.000,B 0.000,C 90.000,E1 41.553} C_DIS
LIN {X 0.163,Y -582.683,Z 1131.022,A 0.000,B 0.000,C 90.000,E1 39.930} C_DIS
LIN {X 0.127,Y -580.719,Z 1131.015,A 0.000,B 0.000,C 90.000,E1 38.588} C_DIS
LIN {X 0.152,Y -578.327,Z 1131.007,A 0.000,B 0.000,C 90.000,E1 37.237} C_DIS
LIN {X -0.170,Y -576.583,Z 1131.002,A 0.000,B 0.000,C 90.000,E1 36.457} C_DIS
LIN {X -0.171,Y -574.586,Z 1130.998,A 0.000,B 0.000,C 90.000,E1 35.644} C_DIS
LIN {X -0.209,Y -573.114,Z 1130.995,A 0.000,B 0.000,C 90.000,E1 35.105} C_DIS
LIN {X 0.020,Y -569.637,Z 1130.989,A 0.000,B 0.000,C 90.000,E1 33.992} C_DIS
LIN {X -0.042,Y -567.655,Z 1130.986,A 0.000,B 0.000,C 90.000,E1 33.452} C_DIS
LIN {X -0.002,Y -564.402,Z 1130.981,A 0.000,B 0.000,C 90.000,E1 32.625} C_DIS
LIN {X 0.098,Y -561.440,Z 1130.977,A 0.000,B 0.000,C 90.000,E1 31.926} C_DIS
LIN {X 0.312,Y -556.079,Z 1130.971,A 0.000,B 0.000,C 90.000,E1 30.797} C_DIS
LIN {X -0.149,Y -549.254,Z 1130.964,A 0.000,B 0.000,C 90.000,E1 29.589} C_DIS
LIN {X 0.117,Y -545.965,Z 1130.961,A 0.000,B 0.000,C 90.000,E1 28.999} C_DIS
LIN {X 0.099,Y -540.582,Z 1130.957,A 0.000,B 0.000,C 90.000,E1 28.153} C_DIS
LIN {X 0.048,Y -536.667,Z 1130.953,A 0.000,B 0.000,C 90.000,E1 27.590} C_DIS
LIN {X 0.075,Y -531.465,Z 1130.949,A 0.000,B 0.000,C 90.000,E1 26.873} C_DIS
LIN {X 0.052,Y -525.862,Z 1130.945,A 0.000,B 0.000,C 90.000,E1 26.155} C_DIS
LIN {X -0.094,Y -521.013,Z 1130.942,A 0.000,B 0.000,C 90.000,E1 25.591} C_DIS
LIN {X 0.156,Y -514.771,Z 1130.938,A 0.000,B 0.000,C 90.000,E1 24.847} C_DIS
LIN {X 0.237,Y -509.453,Z 1130.935,A 0.000,B 0.000,C 90.000,E1 24.259} C_DIS
LIN {X -0.205,Y -501.318,Z 1130.930,A 0.000,B 0.000,C 90.000,E1 23.462} C_DIS
LIN {X -0.211,Y -494.278,Z 1130.926,A 0.000,B 0.000,C 90.000,E1 22.770} C_DIS
LIN {X -0.115,Y -487.138,Z 1130.923,A 0.000,B 0.000,C 90.000,E1 22.078} C_DIS
LIN {X -0.022,Y -479.970,Z 1130.919,A 0.000,B 0.000,C 90.000,E1 21.408} C_DIS
LIN {X 0.110,Y -469.718,Z 1130.914,A 0.000,B 0.000,C 90.000,E1 20.482} C_DIS
LIN {X -0.121,Y -456.272,Z 1130.907,A 0.000,B 0.000,C 90.000,E1 19.322} C_DIS
LIN {X -0.116,Y -437.566,Z 1130.898,A 0.000,B 0.000,C 90.000,E1 17.583} C_DIS
LIN {X 0.077,Y -423.289,Z 1130.889,A 0.000,B 0.000,C 90.000,E1 16.079} C_DIS
LIN {X -0.035,Y -412.211,Z 1130.882,A 0.000,B 0.000,C 90.000,E1 14.828} C_DIS
LIN {X 0.180,Y -403.229,Z 1130.876,A 0.000,B 0.000,C 90.000,E1 13.647} C_DIS
LIN {X 0.165,Y -398.786,Z 1130.872,A 0.000,B 0.000,C 90.000,E1 13.008} C_DIS
LIN {X -0.149,Y -396.768,Z 1130.870,A 0.000,B 0.000,C 90.000,E1 12.703} C_DIS
LIN {X -0.182,Y -394.844,Z 1130.868,A 0.000,B 0.000,C 90.000,E1 12.299} C_DIS
LIN {X -0.154,Y -393.923,Z 1130.867,A 0.000,B 0.000,C 90.000,E1 12.119} C_DIS
LIN {X -0.214,Y -393.285,Z 1130.866,A 0.000,B 0.000,C 90.000,E1 11.951} C_DIS
LIN {X -0.052,Y -392.481,Z 1130.864,A 0.000,B 0.000,C 90.000,E1 11.591} C_DIS
LIN {X 0.200,Y -392.148,Z 1130.861,A 0.000,B 0.000,C 90.000,E1 10.950} C_DIS
LIN {X -0.054,Y -392.794,Z 1130.858,A 0.000,B 0.000,C 90.000,E1 10.366} C_DIS
LIN {X -0.142,Y -394.206,Z 1130.854,A 0.000,B 0.000,C 90.000,E1 9.670} C_DIS
LIN {X 0.005,Y -399.991,Z 1130.842,A 0.000,B 0.000,C 90.000,E1 7.530} C_DIS
LIN {X -0.069,Y -403.757,Z 1130.835,A 0.000,B 0.000,C 90.000,E1 6.315} C_DIS
LIN {X -0.075,Y -405.041,Z 1130.833,A 0.000,B 0.000,C 90.000,E1 5.967} C_DIS
LIN {X -0.097,Y -407.444,Z 1130.830,A 0.000,B 0.000,C 90.000,E1 5.448} C_DIS
LIN {X -0.197,Y -411.796,Z 1130.827,A 0.000,B 0.000,C 90.000,E1 4.878} C_DIS
LIN {X 0.123,Y -413.957,Z 1130.826,A 0.000,B 0.000,C 90.000,E1 4.645} C_DIS
LIN {X -0.017,Y -420.216,Z 1130.823,A 0.000,B 0.000,C 90.000,E1 4.188} C_DIS
LIN {X -0.140,Y -435.962,Z 1130.817,A 0.000,B 0.000,C 90.000,E1 3.094} C_DIS
LIN {X -0.091,Y -460.474,Z 1130.808,A 0.000,B 0.000,C 90.000,E1 1.432} C_DIS
LIN {X -0.204,Y -474.703,Z 1130.803,A 0.000,B 0.000,C 90.000,E1 0.516} C_DIS
LIN {X 0.000,Y -482.049,Z 1130.800,A 0.000,B 0.000,C 90.000,E1 360.000} C_DIS
LIN {X -0.153,Y -491.239,Z 1130.797,A 0.000,B 0.000,C 90.000,E1 359.370} C_DIS
LIN {X -0.182,Y -497.391,Z 1130.794,A 0.000,B 0.000,C 90.000,E1 358.912} C_DIS
LIN {X -0.212,Y -503.304,Z 1130.791,A 0.000,B 0.000,C 90.000,E1 358.453} C_DIS
LIN {X -0.048,Y -510.440,Z 1130.788,A 0.000,B 0.000,C 90.000,E1 357.822} C_DIS
LIN {X -0.033,Y -517.298,Z 1130.784,A 0.000,B 0.000,C 90.000,E1 357.192} C_DIS
LIN {X -0.242,Y -522.618,Z 1130.781,A 0.000,B 0.000,C 90.000,E1 356.674} C_DIS
LIN {X -0.056,Y -528.709,Z 1130.778,A 0.000,B 0.000,C 90.000,E1 355.988} C_DIS
LIN {X 0.219,Y -532.406,Z 1130.775,A 0.000,B 0.000,C 90.000,E1 355.527} C_DIS
LIN {X -0.040,Y -537.900,Z 1130.771,A 0.000,B 0.000,C 90.000,E1 354.837} C_DIS
LIN {X 0.196,Y -541.849,Z 1130.768,A 0.000,B 0.000,C 90.000,E1 354.261} C_DIS
LIN {X -0.186,Y -547.156,Z 1130.764,A 0.000,B 0.000,C 90.000,E1 353.451} C_DIS
LIN {X -0.066,Y -550.428,Z 1130.760,A 0.000,B 0.000,C 90.000,E1 352.875} C_DIS
LIN {X -0.180,Y -554.154,Z 1130.757,A 0.000,B 0.000,C 90.000,E1 352.186} C_DIS
LIN {X 0.064,Y -556.884,Z 1130.753,A 0.000,B 0.000,C 90.000,E1 351.602} C_DIS
LIN {X 0.249,Y -559.350,Z 1130.750,A 0.000,B 0.000,C 90.000,E1 351.027} C_DIS
LIN {X 0.133,Y -562.708,Z 1130.746,A 0.000,B 0.000,C 90.000,E1 350.208} C_DIS
LIN {X -0.206,Y -564.776,Z 1130.743,A 0.000,B 0.000,C 90.000,E1 349.690} C_DIS
LIN {X -0.087,Y -568.603,Z 1130.737,A 0.000,B 0.000,C 90.000,E1 348.578} C_DIS
LIN {X -0.099,Y -571.211,Z 1130.732,A 0.000,B 0.000,C 90.000,E1 347.757} C_DIS
LIN {X -0.245,Y -575.290,Z 1130.724,A 0.000,B 0.000,C 90.000,E1 346.408} C_DIS
LIN {X -0.189,Y -578.978,Z 1130.717,A 0.000,B 0.000,C 90.000,E1 345.046} C_DIS
LIN {X 0.269,Y -581.907,Z 1130.711,A 0.000,B 0.000,C 90.000,E1 343.921} C_DIS
LIN {X -0.289,Y -585.966,Z 1130.702,A 0.000,B 0.000,C 90.000,E1 342.362} C_DIS
LIN {X -0.125,Y -588.475,Z 1130.696,A 0.000,B 0.000,C 90.000,E1 341.275} C_DIS
LIN {X 0.075,Y -590.814,Z 1130.690,A 0.000,B 0.000,C 90.000,E1 340.188} C_DIS
LIN {X 0.186,Y -593.407,Z 1130.683,A 0.000,B 0.000,C 90.000,E1 338.847} C_DIS
LIN {X -0.348,Y -594.870,Z 1130.678,A 0.000,B 0.000,C 90.000,E1 338.103} C_DIS
LIN {X -0.088,Y -596.042,Z 1130.674,A 0.000,B 0.000,C 90.000,E1 337.283} C_DIS
LIN {X -0.216,Y -597.570,Z 1130.667,A 0.000,B 0.000,C 90.000,E1 335.973} C_DIS
LIN {X -0.248,Y -598.404,Z 1130.661,A 0.000,B 0.000,C 90.000,E1 334.921} C_DIS
LIN {X 0.054,Y -598.815,Z 1130.656,A 0.000,B 0.000,C 90.000,E1 334.101} C_DIS
LIN {X 0.089,Y -598.873,Z 1130.652,A 0.000,B 0.000,C 90.000,E1 333.307} C_DIS
LIN {X -0.212,Y -598.502,Z 1130.646,A 0.000,B 0.000,C 90.000,E1 332.281} C_DIS
LIN {X 0.078,Y -597.881,Z 1130.642,A 0.000,B 0.000,C 90.000,E1 331.463} C_DIS
LIN {X 0.201,Y -597.256,Z 1130.639,A 0.000,B 0.000,C 90.000,E1 330.923} C_DIS
LIN {X 0.241,Y -596.057,Z 1130.634,A 0.000,B 0.000,C 90.000,E1 330.127} C_DIS
LIN {X 0.268,Y -594.427,Z 1130.630,A 0.000,B 0.000,C 90.000,E1 329.331} C_DIS
LIN {X 0.277,Y -592.313,Z 1130.625,A 0.000,B 0.000,C 90.000,E1 328.535} C_DIS
LIN {X -0.129,Y -590.602,Z 1130.622,A 0.000,B 0.000,C 90.000,E1 328.043} C_DIS
LIN {X -0.041,Y -588.635,Z 1130.620,A 0.000,B 0.000,C 90.000,E1 327.502} C_DIS
LIN {X 0.032,Y -586.488,Z 1130.617,A 0.000,B 0.000,C 90.000,E1 326.962} C_DIS
LIN {X -0.052,Y -582.797,Z 1130.612,A 0.000,B 0.000,C 90.000,E1 326.167} C_DIS
LIN {X 0.215,Y -579.272,Z 1130.608,A 0.000,B 0.000,C 90.000,E1 325.468} C_DIS
LIN {X 0.002,Y -575.389,Z 1130.605,A 0.000,B 0.000,C 90.000,E1 324.815} C_DIS
LIN {X 0.206,Y -571.062,Z 1130.601,A 0.000,B 0.000,C 90.000,E1 324.116} C_DIS
LIN {X 0.136,Y -567.395,Z 1130.598,A 0.000,B 0.000,C 90.000,E1 323.577} C_DIS
LIN {X -0.304,Y -564.495,Z 1130.595,A 0.000,B 0.000,C 90.000,E1 323.210} C_DIS
LIN {X 0.011,Y -557.988,Z 1130.591,A 0.000,B 0.000,C 90.000,E1 322.351} C_DIS
LIN {X -0.120,Y -548.798,Z 1130.585,A 0.000,B 0.000,C 90.000,E1 321.251} C_DIS
LIN {X -0.219,Y -540.282,Z 1130.579,A 0.000,B 0.000,C 90.000,E1 320.275} C_DIS
LIN {X -0.016,Y -536.529,Z 1130.577,A 0.000,B 0.000,C 90.000,E1 319.828} C_DIS
LIN {X 0.002,Y -534.577,Z 1130.575,A 0.000,B 0.000,C 90.000,E1 319.542} C_DIS
LIN {X -0.065,Y -531.323,Z 1130.572,A 0.000,B 0.000,C 90.000,E1 318.976} C_DIS
LIN {X -0.080,Y -529.976,Z 1130.571,A 0.000,B 0.000,C 90.000,E1 318.690} C_DIS
LIN {X 0.241,Y -528.030,Z 1130.568,A 0.000,B 0.000,C 90.000,E1 318.162} C_DIS
LIN {X -0.216,Y -526.412,Z 1130.565,A 0.000,B 0.000,C 90.000,E1 317.634} C_DIS
LIN {X -0.173,Y -525.247,Z 1130.561,A 0.000,B 0.000,C 90.000,E1 316.905} C_DIS
LIN {X -0.052,Y -524.919,Z 1130.557,A 0.000,B 0.000,C 90.000,E1 316.257} C_DIS
LIN {X -0.105,Y -524.685,Z 1130.555,A 0.000,B 0.000,C 90.000,E1 315.972} C_DIS
LIN {X -0.228,Y -524.628,Z 1130.552,A 0.000,B 0.000,C 90.000,E1 315.405} C_DIS
LIN {X 0.119,Y -525.571,Z 1130.521,A 0.000,B 0.000,C 90.000,E1 309.850} C_DIS
LIN {X 0.216,Y -526.754,Z 1130.510,A 0.000,B 0.000,C 90.000,E1 307.810} C_DIS
LIN {X 0.054,Y -527.866,Z 1130.501,A 0.000,B 0.000,C 90.000,E1 306.091} C_DIS
LIN {X 0.018,Y -529.256,Z 1130.489,A 0.000,B 0.000,C 90.000,E1 304.072} C_DIS
LIN {X 0.007,Y -530.724,Z 1130.478,A 0.000,B 0.000,C 90.000,E1 302.054} C_DIS
LIN {X 0.229,Y -531.832,Z 1130.470,A 0.000,B 0.000,C 90.000,E1 300.590} C_DIS
LIN {X -0.254,Y -532.875,Z 1130.462,A 0.000,B 0.000,C 90.000,E1 299.205} C_DIS
LIN {X 0.221,Y -533.805,Z 1130.454,A 0.000,B 0.000,C 90.000,E1 297.719} C_DIS
LIN {X 0.086,Y -534.219,Z 1130.449,A 0.000,B 0.000,C 90.000,E1 296.873} C_DIS
LIN {X 0.147,Y -534.582,Z 1130.443,A 0.000,B 0.000,C 90.000,E1 295.720} C_DIS
LIN {X -0.219,Y -534.729,Z 1130.438,A 0.000,B 0.000,C 90.000,E1 294.899} C_DIS
LIN {X -0.172,Y -534.788,Z 1130.430,A 0.000,B 0.000,C 90.000,E1 293.462} C_DIS
LIN {X -0.125,Y -534.804,Z 1130.422,A 0.000,B 0.000,C 90.000,E1 292.025} C_DIS
LIN {X -0.079,Y -534.670,Z 1130.413,A 0.000,B 0.000,C 90.000,E1 290.301} C_DIS
LIN {X -0.224,Y -534.408,Z 1130.403,A 0.000,B 0.000,C 90.000,E1 288.598} C_DIS
LIN {X -0.039,Y -533.944,Z 1130.394,A 0.000,B 0.000,C 90.000,E1 286.858} C_DIS
LIN {X -0.094,Y -533.488,Z 1130.387,A 0.000,B 0.000,C 90.000,E1 285.717} C_DIS
LIN {X -0.260,Y -532.818,Z 1130.379,A 0.000,B 0.000,C 90.000,E1 284.300} C_DIS
LIN {X 0.083,Y -532.106,Z 1130.371,A 0.000,B 0.000,C 90.000,E1 282.827} C_DIS
LIN {X -0.179,Y -531.211,Z 1130.362,A 0.000,B 0.000,C 90.000,E1 281.130} C_DIS
LIN {X 0.003,Y -530.074,Z 1130.351,A 0.000,B 0.000,C 90.000,E1 279.095} C_DIS
LIN {X 0.089,Y -529.325,Z 1130.343,A 0.000,B 0.000,C 90.000,E1 277.644} C_DIS
LIN {X 0.108,Y -528.448,Z 1130.333,A 0.000,B 0.000,C 90.000,E1 275.910} C_DIS
LIN {X 0.002,Y -527.716,Z 1130.323,A 0.000,B 0.000,C 90.000,E1 274.188} C_DIS
LIN {X -0.083,Y -527.085,Z 1130.315,A 0.000,B 0.000,C 90.000,E1 272.751} C_DIS
LIN {X -0.244,Y -526.322,Z 1130.306,A 0.000,B 0.000,C 90.000,E1 271.031} C_DIS
LIN {X 0.096,Y -525.512,Z 1130.296,A 0.000,B 0.000,C 90.000,E1 269.255} C_DIS
LIN {X -0.005,Y -525.155,Z 1130.291,A 0.000,B 0.000,C 90.000,E1 268.396} C_DIS
LIN {X -0.184,Y -524.228,Z 1130.281,A 0.000,B 0.000,C 90.000,E1 266.674} C_DIS
LIN {X 0.145,Y -523.226,Z 1130.272,A 0.000,B 0.000,C 90.000,E1 264.894} C_DIS
LIN {X 0.033,Y -522.395,Z 1130.265,A 0.000,B 0.000,C 90.000,E1 263.742} C_DIS
LIN {X -0.176,Y -520.407,Z 1130.254,A 0.000,B 0.000,C 90.000,E1 261.724} C_DIS
LIN {X -0.281,Y -518.654,Z 1130.244,A 0.000,B 0.000,C 90.000,E1 259.982} C_DIS
LIN {X 0.179,Y -517.014,Z 1130.234,A 0.000,B 0.000,C 90.000,E1 258.173} C_DIS
LIN {X 0.203,Y -515.226,Z 1130.225,A 0.000,B 0.000,C 90.000,E1 256.408} C_DIS
LIN {X -0.177,Y -513.654,Z 1130.215,A 0.000,B 0.000,C 90.000,E1 254.685} C_DIS
LIN {X -0.100,Y -511.923,Z 1130.205,A 0.000,B 0.000,C 90.000,E1 252.906} C_DIS
LIN {X 0.125,Y -510.414,Z 1130.197,A 0.000,B 0.000,C 90.000,E1 251.402} C_DIS
LIN {X -0.098,Y -509.139,Z 1130.190,A 0.000,B 0.000,C 90.000,E1 250.242} C_DIS
LIN {X 0.137,Y -507.826,Z 1130.184,A 0.000,B 0.000,C 90.000,E1 249.028} C_DIS
LIN {X 0.158,Y -506.143,Z 1130.175,A 0.000,B 0.000,C 90.000,E1 247.539} C_DIS
LIN {X 0.061,Y -504.663,Z 1130.169,A 0.000,B 0.000,C 90.000,E1 246.357} C_DIS
LIN {X 0.228,Y -502.718,Z 1130.160,A 0.000,B 0.000,C 90.000,E1 244.845} C_DIS
LIN {X -0.098,Y -500.540,Z 1130.152,A 0.000,B 0.000,C 90.000,E1 243.384} C_DIS
LIN {X -0.238,Y -498.313,Z 1130.144,A 0.000,B 0.000,C 90.000,E1 241.897} C_DIS
LIN {X -0.151,Y -495.469,Z 1130.134,A 0.000,B 0.000,C 90.000,E1 240.078} C_DIS
LIN {X -0.059,Y -492.429,Z 1130.124,A 0.000,B 0.000,C 90.000,E1 238.250} C_DIS
LIN {X -0.030,Y -489.391,Z 1130.114,A 0.000,B 0.000,C 90.000,E1 236.421} C_DIS
LIN {X 0.189,Y -486.319,Z 1130.103,A 0.000,B 0.000,C 90.000,E1 234.562} C_DIS
LIN {X 0.181,Y -484.180,Z 1130.096,A 0.000,B 0.000,C 90.000,E1 233.336} C_DIS
LIN {X 0.266,Y -480.448,Z 1130.084,A 0.000,B 0.000,C 90.000,E1 231.170} C_DIS
LIN {X -0.095,Y -477.608,Z 1130.076,A 0.000,B 0.000,C 90.000,E1 229.666} C_DIS
LIN {X 0.047,Y -473.694,Z 1130.064,A 0.000,B 0.000,C 90.000,E1 227.472} C_DIS
LIN {X 0.038,Y -469.835,Z 1130.052,A 0.000,B 0.000,C 90.000,E1 225.283} C_DIS
LIN {X 0.065,Y -465.377,Z 1130.036,A 0.000,B 0.000,C 90.000,E1 222.447} C_DIS
LIN {X -0.070,Y -461.810,Z 1130.022,A 0.000,B 0.000,C 90.000,E1 219.930} C_DIS
LIN {X -0.050,Y -459.767,Z 1130.013,A 0.000,B 0.000,C 90.000,E1 218.338} C_DIS
LIN {X -0.051,Y -457.588,Z 1130.002,A 0.000,B 0.000,C 90.000,E1 216.423} C_DIS
LIN {X -0.116,Y -456.146,Z 1129.995,A 0.000,B 0.000,C 90.000,E1 215.152} C_DIS
LIN {X 0.182,Y -452.642,Z 1129.974,A 0.000,B 0.000,C 90.000,E1 211.258} C_DIS
LIN {X 0.110,Y -451.413,Z 1129.963,A 0.000,B 0.000,C 90.000,E1 209.333} C_DIS
LIN {X 0.142,Y -450.722,Z 1129.949,A 0.000,B 0.000,C 90.000,E1 206.744} C_DIS
LIN {X -0.069,Y -451.198,Z 1129.940,A 0.000,B 0.000,C 90.000,E1 205.155} C_DIS
LIN {X 0.139,Y -452.546,Z 1129.931,A 0.000,B 0.000,C 90.000,E1 203.515} C_DIS
LIN {X 0.194,Y -455.057,Z 1129.922,A 0.000,B 0.000,C 90.000,E1 201.897} C_DIS
LIN {X 0.130,Y -458.277,Z 1129.913,A 0.000,B 0.000,C 90.000,E1 200.301} C_DIS
LIN {X -0.026,Y -462.238,Z 1129.904,A 0.000,B 0.000,C 90.000,E1 198.725} C_DIS
LIN {X 0.066,Y -469.038,Z 1129.892,A 0.000,B 0.000,C 90.000,E1 196.496} C_DIS
LIN {X -0.080,Y -477.726,Z 1129.878,A 0.000,B 0.000,C 90.000,E1 194.008} C_DIS
LIN {X -0.071,Y -487.046,Z 1129.864,A 0.000,B 0.000,C 90.000,E1 191.535} C_DIS
LIN {X -0.216,Y -496.103,Z 1129.851,A 0.000,B 0.000,C 90.000,E1 189.265} C_DIS
LIN {X 0.180,Y -500.410,Z 1129.845,A 0.000,B 0.000,C 90.000,E1 188.163} C_DIS
LIN {X -0.186,Y -505.305,Z 1129.839,A 0.000,B 0.000,C 90.000,E1 187.004} C_DIS
LIN {X -0.147,Y -511.247,Z 1129.831,A 0.000,B 0.000,C 90.000,E1 185.511} C_DIS
LIN {X 0.057,Y -517.221,Z 1129.822,A 0.000,B 0.000,C 90.000,E1 184.012} C_DIS
LIN {X 0.254,Y -524.471,Z 1129.813,A 0.000,B 0.000,C 90.000,E1 182.236} C_DIS
LIN {X 0.089,Y -531.571,Z 1129.803,A 0.000,B 0.000,C 90.000,E1 180.516} C_DIS
LIN {X -0.207,Y -538.154,Z 1129.794,A 0.000,B 0.000,C 90.000,E1 178.969} C_DIS
LIN {X 0.152,Y -543.526,Z 1129.787,A 0.000,B 0.000,C 90.000,E1 177.650} C_DIS
LIN {X -0.064,Y -551.870,Z 1129.776,A 0.000,B 0.000,C 90.000,E1 175.698} C_DIS
LIN {X -0.163,Y -559.015,Z 1129.767,A 0.000,B 0.000,C 90.000,E1 174.033} C_DIS
LIN {X 0.171,Y -567.343,Z 1129.756,A 0.000,B 0.000,C 90.000,E1 172.064} C_DIS
LIN {X -0.038,Y -574.397,Z 1129.747,A 0.000,B 0.000,C 90.000,E1 170.443} C_DIS
LIN {X -0.233,Y -580.097,Z 1129.739,A 0.000,B 0.000,C 90.000,E1 169.106} C_DIS
LIN {X -0.223,Y -585.550,Z 1129.732,A 0.000,B 0.000,C 90.000,E1 167.757} C_DIS
LIN {X -0.116,Y -590.915,Z 1129.724,A 0.000,B 0.000,C 90.000,E1 166.408} C_DIS
LIN {X 0.224,Y -595.951,Z 1129.717,A 0.000,B 0.000,C 90.000,E1 165.046} C_DIS
LIN {X -0.085,Y -598.819,Z 1129.713,A 0.000,B 0.000,C 90.000,E1 164.283} C_DIS
LIN {X -0.209,Y -601.533,Z 1129.708,A 0.000,B 0.000,C 90.000,E1 163.504} C_DIS
LIN {X 0.206,Y -606.683,Z 1129.700,A 0.000,B 0.000,C 90.000,E1 161.891} C_DIS
LIN {X 0.025,Y -610.680,Z 1129.692,A 0.000,B 0.000,C 90.000,E1 160.604} C_DIS
LIN {X -0.032,Y -613.761,Z 1129.687,A 0.000,B 0.000,C 90.000,E1 159.571} C_DIS
LIN {X -0.084,Y -617.305,Z 1129.679,A 0.000,B 0.000,C 90.000,E1 158.284} C_DIS
LIN {X -0.099,Y -621.422,Z 1129.671,A 0.000,B 0.000,C 90.000,E1 156.741} C_DIS
LIN {X -0.365,Y -624.670,Z 1129.664,A 0.000,B 0.000,C 90.000,E1 155.485} C_DIS
END
